LIN {X 0,Y 578.612,Z 1192.309,A -85,B 0,C 180,E1 8897.557,E2 8897.557} C_VEL
LIN {X 0,Y 578.237,Z 1202.22,A -85,B 0,C 180,E1 8901.735,E2 8901.735} C_VEL
LIN {X 0,Y 578.097,Z 1207.67,A -85,B 0,C 180,E1 8905.502,E2 8905.502} C_VEL
LIN {X 0,Y 578.168,Z 1210,A -85,B 0,C 180,E1 8909.999,E2 8909.999} C_VEL
LIN {X 0,Y 578.088,Z 1207.673,A -85,B 0,C 180,E1 8914.497,E2 8914.497} C_VEL
LIN {X 0,Y 578.267,Z 1200.684,A -85,B 0,C 180,E1 8919.02,E2 8919.02} C_VEL
LIN {X 0,Y 578.858,Z 1188.879,A -85,B 0,C 180,E1 8923.588,E2 8923.588} C_VEL
LIN {X 0,Y 580.238,Z 1171.703,A -85,B 0,C 180,E1 8928.21,E2 8928.21} C_VEL
LIN {X 0,Y 582.752,Z 1146.922,A -85,B 0,C 180,E1 8933.18,E2 8933.18} C_VEL
LIN {X 0,Y 586.408,Z 1118.128,A -85,B 0,C 180,E1 8937.635,E2 8937.635} C_VEL
LIN {X 0,Y 591.463,Z 1084.189,A -85,B 0,C 180,E1 8941.799,E2 8941.799} C_VEL
LIN {X 0,Y 597.246,Z 1046.532,A -85,B 0,C 180,E1 8945.448,E2 8945.448} C_VEL
LIN {X 0,Y 603.563,Z 1005.363,A -85,B 0,C 180,E1 8948.616,E2 8948.616} C_VEL
LIN {X 0,Y 609.873,Z 959.425,A -85,B 0,C 180,E1 8951.318,E2 8951.318} C_VEL
LIN {X 0,Y 614.972,Z 913.089,A -85,B 0,C 180,E1 8953.312,E2 8953.312} C_VEL
LIN {X 0,Y 619.146,Z 862.515,A -85,B 0,C 180,E1 8954.794,E2 8954.794} C_VEL
LIN {X 0,Y 620.72,Z 823.615,A -85,B 0,C 180,E1 8955.571,E2 8955.571} C_VEL
LIN {X 0,Y 587.125,Z 766.876,A -85,B 0,C 180,E1 8959.714,E2 8959.714} C_VEL
LIN {X 0,Y 577.318,Z 751.271,A -85,B 0,C 180,E1 8961.134,E2 8961.134} C_VEL
LIN {X 0,Y 577.129,Z 749.56,A -85,B 0,C 180,E1 8961.259,E2 8961.259} C_VEL
LIN {X 0,Y 577.17,Z 749.56,A -85,B 0,C 180,E1 8966.909,E2 8966.909} C_VEL
LIN {X 0,Y 577.189,Z 749.56,A -85,B 0,C 180,E1 8972.89,E2 8972.89} C_VEL
LIN {X 0,Y 577.364,Z 749.56,A -85,B 0,C 180,E1 8978.509,E2 8978.509} C_VEL
LIN {X 0,Y 577.572,Z 749.56,A -85,B 0,C 180,E1 8983.278,E2 8983.278} C_VEL
LIN {X 0,Y 577.694,Z 749.56,A -85,B 0,C 180,E1 8987.925,E2 8987.925} C_VEL
LIN {X 0,Y 577.893,Z 749.56,A -85,B 0,C 180,E1 8993.538,E2 8993.538} C_VEL
LIN {X 0,Y 578.167,Z 749.56,A -85,B 0,C 180,E1 8998.506,E2 8998.506} C_VEL
LIN {X 0,Y 577.98,Z 749.56,A -85,B 0,C 180,E1 9004.503,E2 9004.503} C_VEL
LIN {X 0,Y 577.846,Z 749.56,A -85,B 0,C 180,E1 9009.032,E2 9009.032} C_VEL
LIN {X 0,Y 577.48,Z 749.56,A -85,B 0,C 180,E1 9014.491,E2 9014.491} C_VEL
LIN {X 0,Y 577.308,Z 749.56,A -85,B 0,C 180,E1 9019.899,E2 9019.899} C_VEL
LIN {X 0,Y 577.195,Z 749.56,A -85,B 0,C 180,E1 9024.77,E2 9024.77} C_VEL
LIN {X 0,Y 577.119,Z 749.56,A -85,B 0,C 180,E1 9030.225,E2 9030.225} C_VEL
LIN {X 0,Y 577.219,Z 749.952,A -85,B 0,C 180,E1 9034.568,E2 9034.568} C_VEL
LIN {X 0,Y 579.814,Z 755.423,A -85,B 0,C 180,E1 9034.992,E2 9034.992} C_VEL
LIN {X 0,Y 601.046,Z 789.481,A -85,B 0,C 180,E1 9038.031,E2 9038.031} C_VEL
LIN {X 0,Y 614.345,Z 817.609,A -85,B 0,C 180,E1 9040.099,E2 9040.099} C_VEL
LIN {X 0,Y 610.546,Z 862.835,A -85,B 0,C 180,E1 9041.509,E2 9041.509} C_VEL
LIN {X 0,Y 605.594,Z 905.044,A -85,B 0,C 180,E1 9043.417,E2 9043.417} C_VEL
LIN {X 0,Y 600.085,Z 944.792,A -85,B 0,C 180,E1 9045.805,E2 9045.805} C_VEL
LIN {X 0,Y 593.877,Z 985.069,A -85,B 0,C 180,E1 9049.002,E2 9049.002} C_VEL
LIN {X 0,Y 588.198,Z 1022.822,A -85,B 0,C 180,E1 9052.896,E2 9052.896} C_VEL
LIN {X 0,Y 584.217,Z 1052.857,A -85,B 0,C 180,E1 9056.744,E2 9056.744} C_VEL
LIN {X 0,Y 581.273,Z 1079.147,A -85,B 0,C 180,E1 9061.041,E2 9061.041} C_VEL
LIN {X 0,Y 579.471,Z 1099.154,A -85,B 0,C 180,E1 9065.34,E2 9065.34} C_VEL
LIN {X 0,Y 578.595,Z 1114.303,A -85,B 0,C 180,E1 9069.756,E2 9069.756} C_VEL
LIN {X 0,Y 578.124,Z 1124.044,A -85,B 0,C 180,E1 9074.071,E2 9074.071} C_VEL
LIN {X 0,Y 577.881,Z 1128.776,A -85,B 0,C 180,E1 9077.926,E2 9077.926} C_VEL
LIN {X 0,Y 578.053,Z 1129.657,A -85,B 0,C 180,E1 9082.49,E2 9082.49} C_VEL
LIN {X 0,Y 578.256,Z 1125.379,A -85,B 0,C 180,E1 9087.005,E2 9087.005} C_VEL
LIN {X 0,Y 578.486,Z 1116.064,A -85,B 0,C 180,E1 9091.498,E2 9091.498} C_VEL
LIN {X 0,Y 579.246,Z 1102.955,A -85,B 0,C 180,E1 9095.615,E2 9095.615} C_VEL
LIN {X 0,Y 580.791,Z 1083.025,A -85,B 0,C 180,E1 9100.116,E2 9100.116} C_VEL
LIN {X 0,Y 583.365,Z 1059.112,A -85,B 0,C 180,E1 9104.247,E2 9104.247} C_VEL
LIN {X 0,Y 587.673,Z 1026.88,A -85,B 0,C 180,E1 9108.555,E2 9108.555} C_VEL
LIN {X 0,Y 593.59,Z 986.738,A -85,B 0,C 180,E1 9112.746,E2 9112.746} C_VEL
LIN {X 0,Y 599.698,Z 946.386,A -85,B 0,C 180,E1 9115.968,E2 9115.968} C_VEL
LIN {X 0,Y 605.16,Z 906.666,A -85,B 0,C 180,E1 9118.383,E2 9118.383} C_VEL
LIN {X 0,Y 610.26,Z 863.781,A -85,B 0,C 180,E1 9120.324,E2 9120.324} C_VEL
LIN {X 0,Y 613.896,Z 820.422,A -85,B 0,C 180,E1 9121.706,E2 9121.706} C_VEL
LIN {X 0,Y 612.931,Z 814.925,A -85,B 0,C 180,E1 9121.963,E2 9121.963} C_VEL
LIN {X 0,Y 599.509,Z 787.876,A -85,B 0,C 180,E1 9123.901,E2 9123.901} C_VEL
LIN {X 0,Y 577.285,Z 750.933,A -85,B 0,C 180,E1 9126.769,E2 9126.769} C_VEL
LIN {X 0,Y 577.172,Z 749.56,A -85,B 0,C 180,E1 9126.863,E2 9126.863} C_VEL
LIN {X 0,Y 577.186,Z 749.56,A -85,B 0,C 180,E1 9132.9,E2 9132.9} C_VEL
LIN {X 0,Y 577.153,Z 749.56,A -85,B 0,C 180,E1 9139.107,E2 9139.107} C_VEL
LIN {X 0,Y 577.103,Z 749.56,A -85,B 0,C 180,E1 9144.82,E2 9144.82} C_VEL
LIN {X 0,Y 577.103,Z 749.56,A -85,B 0,C 180,E1 9150.159,E2 9150.159} C_VEL
LIN {X 0,Y 577.201,Z 749.56,A -85,B 0,C 180,E1 9155.231,E2 9155.231} C_VEL
LIN {X 0,Y 577.331,Z 749.56,A -85,B 0,C 180,E1 9160.44,E2 9160.44} C_VEL
LIN {X 0,Y 577.534,Z 749.56,A -85,B 0,C 180,E1 9166.375,E2 9166.375} C_VEL
LIN {X 0,Y 577.842,Z 749.56,A -85,B 0,C 180,E1 9170.968,E2 9170.968} C_VEL
LIN {X 0,Y 578.111,Z 749.56,A -85,B 0,C 180,E1 9176.999,E2 9176.999} C_VEL
LIN {X 0,Y 578.183,Z 749.56,A -85,B 0,C 180,E1 9181.494,E2 9181.494} C_VEL
LIN {X 0,Y 577.908,Z 749.56,A -85,B 0,C 180,E1 9187.508,E2 9187.508} C_VEL
LIN {X 0,Y 577.699,Z 749.56,A -85,B 0,C 180,E1 9193.612,E2 9193.612} C_VEL
LIN {X 0,Y 577.611,Z 749.56,A -85,B 0,C 180,E1 9198.293,E2 9198.293} C_VEL
LIN {X 0,Y 577.4,Z 749.56,A -85,B 0,C 180,E1 9203.651,E2 9203.651} C_VEL
LIN {X 0,Y 577.382,Z 749.56,A -85,B 0,C 180,E1 9208.102,E2 9208.102} C_VEL
LIN {X 0,Y 577.242,Z 749.56,A -85,B 0,C 180,E1 9213.346,E2 9213.346} C_VEL
LIN {X 0,Y 577.164,Z 749.56,A -85,B 0,C 180,E1 9218.983,E2 9218.983} C_VEL
LIN {X 0,Y 579.391,Z 755.018,A -85,B 0,C 180,E1 9219.32,E2 9219.32} C_VEL
LIN {X 0,Y 610.577,Z 806.083,A -85,B 0,C 180,E1 9223.218,E2 9223.218} C_VEL
LIN {X 0,Y 621.286,Z 825.092,A -85,B 0,C 180,E1 9224.485,E2 9224.485} C_VEL
LIN {X 0,Y 618.48,Z 874.739,A -85,B 0,C 180,E1 9225.498,E2 9225.498} C_VEL
LIN {X 0,Y 614.01,Z 922.392,A -85,B 0,C 180,E1 9227.039,E2 9227.039} C_VEL
LIN {X 0,Y 613.212,Z 931.376,A -85,B 0,C 180,E1 9227.398,E2 9227.398} C_VEL
LIN {X 0,Y 608.294,Z 947.479,A -85,B 0,C 180,E1 9227.866,E2 9227.866} C_VEL
LIN {X 0,Y 603.135,Z 963.24,A -85,B 0,C 180,E1 9228.403,E2 9228.403} C_VEL
LIN {X 0,Y 597.496,Z 1003.581,A -85,B 0,C 180,E1 9230.781,E2 9230.781} C_VEL
LIN {X 0,Y 591.158,Z 1043.01,A -85,B 0,C 180,E1 9233.785,E2 9233.785} C_VEL
LIN {X 0,Y 584.765,Z 1082.334,A -85,B 0,C 180,E1 9237.573,E2 9237.573} C_VEL
LIN {X 0,Y 579.229,Z 1116.9,A -85,B 0,C 180,E1 9241.815,E2 9241.815} C_VEL
LIN {X 0,Y 575.32,Z 1145.203,A -85,B 0,C 180,E1 9246.181,E2 9246.181} C_VEL
LIN {X 0,Y 572.667,Z 1168.231,A -85,B 0,C 180,E1 9250.74,E2 9250.74} C_VEL
LIN {X 0,Y 571.23,Z 1186.567,A -85,B 0,C 180,E1 9255.501,E2 9255.501} C_VEL
LIN {X 0,Y 570.523,Z 1199.103,A -85,B 0,C 180,E1 9260.086,E2 9260.086} C_VEL
LIN {X 0,Y 570.308,Z 1205.908,A -85,B 0,C 180,E1 9263.915,E2 9263.915} C_VEL
LIN {X 0,Y 570.149,Z 1209.667,A -85,B 0,C 180,E1 9268.48,E2 9268.48} C_VEL
LIN {X 0,Y 570.3,Z 1208.914,A -85,B 0,C 180,E1 9273.037,E2 9273.037} C_VEL
LIN {X 0,Y 570.311,Z 1203.554,A -85,B 0,C 180,E1 9277.612,E2 9277.612} C_VEL
LIN {X 0,Y 570.709,Z 1193.421,A -85,B 0,C 180,E1 9282.229,E2 9282.229} C_VEL
LIN {X 0,Y 571.785,Z 1178.004,A -85,B 0,C 180,E1 9286.9,E2 9286.9} C_VEL
LIN {X 0,Y 573.906,Z 1156.975,A -85,B 0,C 180,E1 9291.63,E2 9291.63} C_VEL
LIN {X 0,Y 577.264,Z 1130.743,A -85,B 0,C 180,E1 9296.17,E2 9296.17} C_VEL
LIN {X 0,Y 582.138,Z 1098.258,A -85,B 0,C 180,E1 9300.604,E2 9300.604} C_VEL
LIN {X 0,Y 588.075,Z 1061.38,A -85,B 0,C 180,E1 9304.559,E2 9304.559} C_VEL
LIN {X 0,Y 594.538,Z 1021.722,A -85,B 0,C 180,E1 9307.94,E2 9307.94} C_VEL
LIN {X 0,Y 601.245,Z 978.007,A -85,B 0,C 180,E1 9310.802,E2 9310.802} C_VEL
LIN {X 0,Y 606.913,Z 932.395,A -85,B 0,C 180,E1 9313.024,E2 9313.024} C_VEL
LIN {X 0,Y 611.296,Z 887.394,A -85,B 0,C 180,E1 9314.618,E2 9314.618} C_VEL
LIN {X 0,Y 614.809,Z 838.477,A -85,B 0,C 180,E1 9315.774,E2 9315.774} C_VEL
LIN {X 0,Y 614.638,Z 826.617,A -85,B 0,C 180,E1 9316.032,E2 9316.032} C_VEL
LIN {X 0,Y 582.329,Z 771.526,A -85,B 0,C 180,E1 9320.165,E2 9320.165} C_VEL
LIN {X 0,Y 571.112,Z 754.658,A -85,B 0,C 180,E1 9321.827,E2 9321.827} C_VEL
LIN {X 0,Y 569.234,Z 749.56,A -85,B 0,C 180,E1 9322.219,E2 9322.219} C_VEL
LIN {X 0,Y 569.252,Z 749.56,A -85,B 0,C 180,E1 9328.152,E2 9328.152} C_VEL
LIN {X 0,Y 569.31,Z 749.56,A -85,B 0,C 180,E1 9333.181,E2 9333.181} C_VEL
LIN {X 0,Y 569.446,Z 749.56,A -85,B 0,C 180,E1 9338.245,E2 9338.245} C_VEL
LIN {X 0,Y 569.635,Z 749.56,A -85,B 0,C 180,E1 9343.038,E2 9343.038} C_VEL
LIN {X 0,Y 569.819,Z 749.56,A -85,B 0,C 180,E1 9348.874,E2 9348.874} C_VEL
LIN {X 0,Y 570.05,Z 749.56,A -85,B 0,C 180,E1 9353.917,E2 9353.917} C_VEL
LIN {X 0,Y 570.266,Z 749.56,A -85,B 0,C 180,E1 9360.004,E2 9360.004} C_VEL
LIN {X 0,Y 570.07,Z 749.56,A -85,B 0,C 180,E1 9364.565,E2 9364.565} C_VEL
LIN {X 0,Y 569.921,Z 749.56,A -85,B 0,C 180,E1 9369.158,E2 9369.158} C_VEL
LIN {X 0,Y 569.615,Z 749.56,A -85,B 0,C 180,E1 9373.818,E2 9373.818} C_VEL
LIN {X 0,Y 569.384,Z 749.56,A -85,B 0,C 180,E1 9378.576,E2 9378.576} C_VEL
LIN {X 0,Y 569.302,Z 749.56,A -85,B 0,C 180,E1 9383.468,E2 9383.468} C_VEL
LIN {X 0,Y 569.204,Z 749.56,A -85,B 0,C 180,E1 9388.828,E2 9388.828} C_VEL
LIN {X 0,Y 569.282,Z 749.594,A -85,B 0,C 180,E1 9393.55,E2 9393.55} C_VEL
LIN {X 0,Y 571.523,Z 755.068,A -85,B 0,C 180,E1 9393.95,E2 9393.95} C_VEL
LIN {X 0,Y 589.479,Z 782.711,A -85,B 0,C 180,E1 9396.648,E2 9396.648} C_VEL
LIN {X 0,Y 605.75,Z 813.927,A -85,B 0,C 180,E1 9399.164,E2 9399.164} C_VEL
LIN {X 0,Y 608.425,Z 822.45,A -85,B 0,C 180,E1 9399.699,E2 9399.699} C_VEL
LIN {X 0,Y 604.318,Z 866.169,A -85,B 0,C 180,E1 9401.115,E2 9401.115} C_VEL
LIN {X 0,Y 598.886,Z 910.311,A -85,B 0,C 180,E1 9403.176,E2 9403.176} C_VEL
LIN {X 0,Y 592.946,Z 950.211,A -85,B 0,C 180,E1 9405.687,E2 9405.687} C_VEL
LIN {X 0,Y 586.591,Z 989.264,A -85,B 0,C 180,E1 9408.889,E2 9408.889} C_VEL
LIN {X 0,Y 580.689,Z 1025.536,A -85,B 0,C 180,E1 9412.786,E2 9412.786} C_VEL
LIN {X 0,Y 575.878,Z 1059.375,A -85,B 0,C 180,E1 9417.383,E2 9417.383} C_VEL
LIN {X 0,Y 573.067,Z 1083.698,A -85,B 0,C 180,E1 9421.665,E2 9421.665} C_VEL
LIN {X 0,Y 571.421,Z 1103.026,A -85,B 0,C 180,E1 9426.107,E2 9426.107} C_VEL
LIN {X 0,Y 570.606,Z 1117.129,A -85,B 0,C 180,E1 9430.693,E2 9430.693} C_VEL
LIN {X 0,Y 570.191,Z 1125.995,A -85,B 0,C 180,E1 9435.211,E2 9435.211} C_VEL
LIN {X 0,Y 569.984,Z 1129.637,A -85,B 0,C 180,E1 9439.306,E2 9439.306} C_VEL
LIN {X 0,Y 570.162,Z 1128.85,A -85,B 0,C 180,E1 9443.915,E2 9443.915} C_VEL
LIN {X 0,Y 570.299,Z 1123.147,A -85,B 0,C 180,E1 9448.482,E2 9448.482} C_VEL
LIN {X 0,Y 570.789,Z 1113.278,A -85,B 0,C 180,E1 9452.656,E2 9452.656} C_VEL
LIN {X 0,Y 571.884,Z 1097.491,A -85,B 0,C 180,E1 9457.211,E2 9457.211} C_VEL
LIN {X 0,Y 574.022,Z 1075.686,A -85,B 0,C 180,E1 9461.773,E2 9461.773} C_VEL
LIN {X 0,Y 577.236,Z 1049.762,A -85,B 0,C 180,E1 9465.955,E2 9465.955} C_VEL
LIN {X 0,Y 582.581,Z 1013.881,A -85,B 0,C 180,E1 9470.477,E2 9470.477} C_VEL
LIN {X 0,Y 588.507,Z 977.222,A -85,B 0,C 180,E1 9474.072,E2 9474.072} C_VEL
LIN {X 0,Y 594.407,Z 938.894,A -85,B 0,C 180,E1 9476.981,E2 9476.981} C_VEL
LIN {X 0,Y 600.477,Z 895.788,A -85,B 0,C 180,E1 9479.464,E2 9479.464} C_VEL
LIN {X 0,Y 605.681,Z 850.137,A -85,B 0,C 180,E1 9481.335,E2 9481.335} C_VEL
LIN {X 0,Y 607.753,Z 819.864,A -85,B 0,C 180,E1 9482.278,E2 9482.278} C_VEL
LIN {X 0,Y 595.074,Z 793.605,A -85,B 0,C 180,E1 9484.196,E2 9484.196} C_VEL
LIN {X 0,Y 569.437,Z 751.318,A -85,B 0,C 180,E1 9487.595,E2 9487.595} C_VEL
LIN {X 0,Y 569.233,Z 749.56,A -85,B 0,C 180,E1 9487.784,E2 9487.784} C_VEL
LIN {X 0,Y 569.194,Z 749.56,A -85,B 0,C 180,E1 9493.652,E2 9493.652} C_VEL
LIN {X 0,Y 569.167,Z 749.56,A -85,B 0,C 180,E1 9498.407,E2 9498.407} C_VEL
LIN {X 0,Y 569.217,Z 749.56,A -85,B 0,C 180,E1 9504.258,E2 9504.258} C_VEL
LIN {X 0,Y 569.192,Z 749.56,A -85,B 0,C 180,E1 9509.701,E2 9509.701} C_VEL
LIN {X 0,Y 569.248,Z 749.56,A -85,B 0,C 180,E1 9514.861,E2 9514.861} C_VEL
LIN {X 0,Y 569.364,Z 749.56,A -85,B 0,C 180,E1 9519.812,E2 9519.812} C_VEL
LIN {X 0,Y 569.496,Z 749.56,A -85,B 0,C 180,E1 9524.608,E2 9524.608} C_VEL
LIN {X 0,Y 569.819,Z 749.56,A -85,B 0,C 180,E1 9529.297,E2 9529.297} C_VEL
LIN {X 0,Y 570.017,Z 749.56,A -85,B 0,C 180,E1 9533.908,E2 9533.908} C_VEL
LIN {X 0,Y 570.138,Z 749.56,A -85,B 0,C 180,E1 9538.477,E2 9538.477} C_VEL
LIN {X 0,Y 570.069,Z 749.56,A -85,B 0,C 180,E1 9543.035,E2 9543.035} C_VEL
LIN {X 0,Y 569.99,Z 749.56,A -85,B 0,C 180,E1 9547.613,E2 9547.613} C_VEL
LIN {X 0,Y 569.785,Z 749.56,A -85,B 0,C 180,E1 9553.805,E2 9553.805} C_VEL
LIN {X 0,Y 569.686,Z 749.56,A -85,B 0,C 180,E1 9558.557,E2 9558.557} C_VEL
LIN {X 0,Y 569.509,Z 749.56,A -85,B 0,C 180,E1 9563.45,E2 9563.45} C_VEL
LIN {X 0,Y 569.389,Z 749.56,A -85,B 0,C 180,E1 9568.858,E2 9568.858} C_VEL
LIN {X 0,Y 569.253,Z 749.56,A -85,B 0,C 180,E1 9574.621,E2 9574.621} C_VEL
LIN {X 0,Y 569.31,Z 750.309,A -85,B 0,C 180,E1 9578.161,E2 9578.161} C_VEL
LIN {X 0,Y 572.281,Z 755.784,A -85,B 0,C 180,E1 9578.584,E2 9578.584} C_VEL
LIN {X 0,Y 606.158,Z 811.799,A -85,B 0,C 180,E1 9582.908,E2 9582.908} C_VEL
LIN {X 0,Y 615.297,Z 827.805,A -85,B 0,C 180,E1 9584.02,E2 9584.02} C_VEL
LIN {X 0,Y 612.316,Z 876.778,A -85,B 0,C 180,E1 9585.064,E2 9585.064} C_VEL
LIN {X 0,Y 607.591,Z 924.963,A -85,B 0,C 180,E1 9586.663,E2 9586.663} C_VEL
LIN {X 0,Y 603.135,Z 963.24,A -85,B 0,C 180,E1 9588.403,E2 9588.403} C_VEL
LIN {X 0,Y 598,Z 978.76,A -85,B 0,C 180,E1 9589.009,E2 9589.009} C_VEL
LIN {X 0,Y 592.579,Z 993.901,A -85,B 0,C 180,E1 9589.68,E2 9589.68} C_VEL
LIN {X 0,Y 586.197,Z 1032.86,A -85,B 0,C 180,E1 9592.455,E2 9592.455} C_VEL
LIN {X 0,Y 579.745,Z 1070.845,A -85,B 0,C 180,E1 9595.915,E2 9595.915} C_VEL
LIN {X 0,Y 573.522,Z 1107.345,A -85,B 0,C 180,E1 9600.13,E2 9600.13} C_VEL
LIN {X 0,Y 569.067,Z 1136.294,A -85,B 0,C 180,E1 9604.343,E2 9604.343} C_VEL
LIN {X 0,Y 565.606,Z 1162.666,A -85,B 0,C 180,E1 9609.235,E2 9609.235} C_VEL
LIN {X 0,Y 563.725,Z 1181.011,A -85,B 0,C 180,E1 9613.652,E2 9613.652} C_VEL
LIN {X 0,Y 562.769,Z 1195.153,A -85,B 0,C 180,E1 9618.284,E2 9618.284} C_VEL
LIN {X 0,Y 562.455,Z 1204.876,A -85,B 0,C 180,E1 9623.133,E2 9623.133} C_VEL
LIN {X 0,Y 562.361,Z 1208.909,A -85,B 0,C 180,E1 9626.919,E2 9626.919} C_VEL
LIN {X 0,Y 562.506,Z 1209.667,A -85,B 0,C 180,E1 9631.539,E2 9631.539} C_VEL
LIN {X 0,Y 562.41,Z 1205.831,A -85,B 0,C 180,E1 9636.23,E2 9636.23} C_VEL
LIN {X 0,Y 562.718,Z 1197.317,A -85,B 0,C 180,E1 9640.834,E2 9640.834} C_VEL
LIN {X 0,Y 563.546,Z 1183.708,A -85,B 0,C 180,E1 9645.553,E2 9645.553} C_VEL
LIN {X 0,Y 565.132,Z 1166.494,A -85,B 0,C 180,E1 9649.933,E2 9649.933} C_VEL
LIN {X 0,Y 568.012,Z 1142.832,A -85,B 0,C 180,E1 9654.562,E2 9654.562} C_VEL
LIN {X 0,Y 572.688,Z 1112.559,A -85,B 0,C 180,E1 9659.18,E2 9659.18} C_VEL
LIN {X 0,Y 578.359,Z 1078.518,A -85,B 0,C 180,E1 9663.276,E2 9663.276} C_VEL
LIN {X 0,Y 585.156,Z 1039.262,A -85,B 0,C 180,E1 9667.024,E2 9667.024} C_VEL
LIN {X 0,Y 591.517,Z 1000.569,A -85,B 0,C 180,E1 9669.905,E2 9669.905} C_VEL
LIN {X 0,Y 597.952,Z 953.868,A -85,B 0,C 180,E1 9672.532,E2 9672.532} C_VEL
LIN {X 0,Y 603.268,Z 906.93,A -85,B 0,C 180,E1 9674.488,E2 9674.488} C_VEL
LIN {X 0,Y 607.841,Z 855.273,A -85,B 0,C 180,E1 9675.951,E2 9675.951} C_VEL
LIN {X 0,Y 609.068,Z 830.48,A -85,B 0,C 180,E1 9676.444,E2 9676.444} C_VEL
LIN {X 0,Y 577.572,Z 776.18,A -85,B 0,C 180,E1 9680.624,E2 9680.624} C_VEL
LIN {X 0,Y 563.661,Z 755.147,A -85,B 0,C 180,E1 9682.777,E2 9682.777} C_VEL
LIN {X 0,Y 561.297,Z 749.56,A -85,B 0,C 180,E1 9683.323,E2 9683.323} C_VEL
LIN {X 0,Y 561.314,Z 749.56,A -85,B 0,C 180,E1 9689.482,E2 9689.482} C_VEL
LIN {X 0,Y 561.42,Z 749.56,A -85,B 0,C 180,E1 9694.495,E2 9694.495} C_VEL
LIN {X 0,Y 561.587,Z 749.56,A -85,B 0,C 180,E1 9700.351,E2 9700.351} C_VEL
LIN {X 0,Y 561.838,Z 749.56,A -85,B 0,C 180,E1 9705.996,E2 9705.996} C_VEL
LIN {X 0,Y 562.005,Z 749.56,A -85,B 0,C 180,E1 9710.72,E2 9710.72} C_VEL
LIN {X 0,Y 562.189,Z 749.56,A -85,B 0,C 180,E1 9715.379,E2 9715.379} C_VEL
LIN {X 0,Y 562.365,Z 749.56,A -85,B 0,C 180,E1 9720.004,E2 9720.004} C_VEL
LIN {X 0,Y 562.159,Z 749.56,A -85,B 0,C 180,E1 9724.63,E2 9724.63} C_VEL
LIN {X 0,Y 562.006,Z 749.56,A -85,B 0,C 180,E1 9729.289,E2 9729.289} C_VEL
LIN {X 0,Y 561.66,Z 749.56,A -85,B 0,C 180,E1 9734.407,E2 9734.407} C_VEL
LIN {X 0,Y 561.446,Z 749.56,A -85,B 0,C 180,E1 9740.486,E2 9740.486} C_VEL
LIN {X 0,Y 561.357,Z 749.56,A -85,B 0,C 180,E1 9745.518,E2 9745.518} C_VEL
LIN {X 0,Y 561.29,Z 749.56,A -85,B 0,C 180,E1 9751.526,E2 9751.526} C_VEL
LIN {X 0,Y 561.297,Z 749.56,A -85,B 0,C 180,E1 9752.472,E2 9752.472} C_VEL
LIN {X 0,Y 563.51,Z 755.009,A -85,B 0,C 180,E1 9752.89,E2 9752.89} C_VEL
LIN {X 0,Y 577.76,Z 775.916,A -85,B 0,C 180,E1 9755.134,E2 9755.134} C_VEL
LIN {X 0,Y 595.276,Z 806.94,A -85,B 0,C 180,E1 9757.886,E2 9757.886} C_VEL
LIN {X 0,Y 602.732,Z 824.081,A -85,B 0,C 180,E1 9759.2,E2 9759.2} C_VEL
LIN {X 0,Y 598.408,Z 867.609,A -85,B 0,C 180,E1 9760.636,E2 9760.636} C_VEL
LIN {X 0,Y 592.864,Z 910.622,A -85,B 0,C 180,E1 9762.665,E2 9762.665} C_VEL
LIN {X 0,Y 586.622,Z 950.54,A -85,B 0,C 180,E1 9765.188,E2 9765.188} C_VEL
LIN {X 0,Y 580.114,Z 988.793,A -85,B 0,C 180,E1 9768.338,E2 9768.338} C_VEL
LIN {X 0,Y 573.941,Z 1024.495,A -85,B 0,C 180,E1 9772.182,E2 9772.182} C_VEL
LIN {X 0,Y 568.989,Z 1055.093,A -85,B 0,C 180,E1 9776.407,E2 9776.407} C_VEL
LIN {X 0,Y 565.873,Z 1079.951,A -85,B 0,C 180,E1 9780.63,E2 9780.63} C_VEL
LIN {X 0,Y 563.785,Z 1100.396,A -85,B 0,C 180,E1 9785.218,E2 9785.218} C_VEL
LIN {X 0,Y 562.873,Z 1114.699,A -85,B 0,C 180,E1 9789.574,E2 9789.574} C_VEL
LIN {X 0,Y 562.349,Z 1124.877,A -85,B 0,C 180,E1 9794.413,E2 9794.413} C_VEL
LIN {X 0,Y 562.087,Z 1129.608,A -85,B 0,C 180,E1 9799.154,E2 9799.154} C_VEL
LIN {X 0,Y 562.254,Z 1128.822,A -85,B 0,C 180,E1 9803.998,E2 9803.998} C_VEL
LIN {X 0,Y 562.403,Z 1123.372,A -85,B 0,C 180,E1 9808.461,E2 9808.461} C_VEL
LIN {X 0,Y 562.902,Z 1113.654,A -85,B 0,C 180,E1 9812.693,E2 9812.693} C_VEL
LIN {X 0,Y 564.07,Z 1097.98,A -85,B 0,C 180,E1 9817.315,E2 9817.315} C_VEL
LIN {X 0,Y 566.182,Z 1077.441,A -85,B 0,C 180,E1 9821.743,E2 9821.743} C_VEL
LIN {X 0,Y 569.857,Z 1049.36,A -85,B 0,C 180,E1 9826.365,E2 9826.365} C_VEL
LIN {X 0,Y 575.388,Z 1015.913,A -85,B 0,C 180,E1 9830.731,E2 9830.731} C_VEL
LIN {X 0,Y 581.602,Z 979.378,A -85,B 0,C 180,E1 9834.383,E2 9834.383} C_VEL
LIN {X 0,Y 587.752,Z 941.688,A -85,B 0,C 180,E1 9837.312,E2 9837.312} C_VEL
LIN {X 0,Y 594.335,Z 897.041,A -85,B 0,C 180,E1 9839.928,E2 9839.928} C_VEL
LIN {X 0,Y 599.696,Z 852.103,A -85,B 0,C 180,E1 9841.79,E2 9841.79} C_VEL
LIN {X 0,Y 601.685,Z 822.463,A -85,B 0,C 180,E1 9842.75,E2 9842.75} C_VEL
LIN {X 0,Y 587.274,Z 793.511,A -85,B 0,C 180,E1 9844.954,E2 9844.954} C_VEL
LIN {X 0,Y 561.404,Z 750.508,A -85,B 0,C 180,E1 9848.496,E2 9848.496} C_VEL
LIN {X 0,Y 561.343,Z 749.56,A -85,B 0,C 180,E1 9848.669,E2 9848.669} C_VEL
LIN {X 0,Y 561.299,Z 749.56,A -85,B 0,C 180,E1 9854.426,E2 9854.426} C_VEL
LIN {X 0,Y 561.223,Z 749.56,A -85,B 0,C 180,E1 9859.736,E2 9859.736} C_VEL
LIN {X 0,Y 561.294,Z 749.56,A -85,B 0,C 180,E1 9865.566,E2 9865.566} C_VEL
LIN {X 0,Y 561.264,Z 749.56,A -85,B 0,C 180,E1 9871.006,E2 9871.006} C_VEL
LIN {X 0,Y 561.376,Z 749.56,A -85,B 0,C 180,E1 9876.239,E2 9876.239} C_VEL
LIN {X 0,Y 561.448,Z 749.56,A -85,B 0,C 180,E1 9881.152,E2 9881.152} C_VEL
LIN {X 0,Y 561.671,Z 749.56,A -85,B 0,C 180,E1 9885.983,E2 9885.983} C_VEL
LIN {X 0,Y 562.005,Z 749.56,A -85,B 0,C 180,E1 9890.711,E2 9890.711} C_VEL
LIN {X 0,Y 562.293,Z 749.56,A -85,B 0,C 180,E1 9896.915,E2 9896.915} C_VEL
LIN {X 0,Y 562.368,Z 749.56,A -85,B 0,C 180,E1 9901.536,E2 9901.536} C_VEL
LIN {X 0,Y 562.08,Z 749.56,A -85,B 0,C 180,E1 9907.721,E2 9907.721} C_VEL
LIN {X 0,Y 561.884,Z 749.56,A -85,B 0,C 180,E1 9912.42,E2 9912.42} C_VEL
LIN {X 0,Y 561.816,Z 749.56,A -85,B 0,C 180,E1 9917.206,E2 9917.206} C_VEL
LIN {X 0,Y 561.638,Z 749.56,A -85,B 0,C 180,E1 9922.124,E2 9922.124} C_VEL
LIN {X 0,Y 561.528,Z 749.56,A -85,B 0,C 180,E1 9927.368,E2 9927.368} C_VEL
LIN {X 0,Y 561.35,Z 749.56,A -85,B 0,C 180,E1 9932.57,E2 9932.57} C_VEL
LIN {X 0,Y 561.38,Z 749.56,A -85,B 0,C 180,E1 9937.265,E2 9937.265} C_VEL
LIN {X 0,Y 563.756,Z 755.23,A -85,B 0,C 180,E1 9937.642,E2 9937.642} C_VEL
LIN {X 0,Y 594.417,Z 804.941,A -85,B 0,C 180,E1 9941.684,E2 9941.684} C_VEL
LIN {X 0,Y 609.445,Z 831.101,A -85,B 0,C 180,E1 9943.566,E2 9943.566} C_VEL
LIN {X 0,Y 605.951,Z 881.237,A -85,B 0,C 180,E1 9944.691,E2 9944.691} C_VEL
LIN {X 0,Y 601.062,Z 928.661,A -85,B 0,C 180,E1 9946.323,E2 9946.323} C_VEL
LIN {X 0,Y 595.175,Z 974.72,A -85,B 0,C 180,E1 9948.542,E2 9948.542} C_VEL
LIN {X 0,Y 592.579,Z 993.901,A -85,B 0,C 180,E1 9949.68,E2 9949.68} C_VEL
LIN {X 0,Y 586.992,Z 1008.779,A -85,B 0,C 180,E1 9950.406,E2 9950.406} C_VEL
LIN {X 0,Y 581.298,Z 1023.202,A -85,B 0,C 180,E1 9951.206,E2 9951.206} C_VEL
LIN {X 0,Y 574.745,Z 1060.533,A -85,B 0,C 180,E1 9954.428,E2 9954.428} C_VEL
LIN {X 0,Y 568.08,Z 1097.562,A -85,B 0,C 180,E1 9958.457,E2 9958.457} C_VEL
LIN {X 0,Y 562.494,Z 1130.449,A -85,B 0,C 180,E1 9963.041,E2 9963.041} C_VEL
LIN {X 0,Y 558.657,Z 1156.976,A -85,B 0,C 180,E1 9967.747,E2 9967.747} C_VEL
LIN {X 0,Y 556.326,Z 1177.995,A -85,B 0,C 180,E1 9972.614,E2 9972.614} C_VEL
LIN {X 0,Y 555.018,Z 1193.416,A -85,B 0,C 180,E1 9977.419,E2 9977.419} C_VEL
LIN {X 0,Y 554.547,Z 1203.545,A -85,B 0,C 180,E1 9982.168,E2 9982.168} C_VEL
LIN {X 0,Y 554.466,Z 1208.906,A -85,B 0,C 180,E1 9986.875,E2 9986.875} C_VEL
LIN {X 0,Y 554.627,Z 1209.667,A -85,B 0,C 180,E1 9991.56,E2 9991.56} C_VEL
LIN {X 0,Y 554.538,Z 1205.911,A -85,B 0,C 180,E1 9996.257,E2 9996.257} C_VEL
LIN {X 0,Y 554.841,Z 1197.314,A -85,B 0,C 180,E1 10000.99,E2 10000.99} C_VEL
LIN {X 0,Y 555.71,Z 1183.707,A -85,B 0,C 180,E1 10005.778,E2 10005.778} C_VEL
LIN {X 0,Y 557.686,Z 1164.736,A -85,B 0,C 180,E1 10010.624,E2 10010.624} C_VEL
LIN {X 0,Y 560.834,Z 1140.431,A -85,B 0,C 180,E1 10015.323,E2 10015.323} C_VEL
LIN {X 0,Y 565.905,Z 1109.977,A -85,B 0,C 180,E1 10019.949,E2 10019.949} C_VEL
LIN {X 0,Y 572.134,Z 1074.771,A -85,B 0,C 180,E1 10024.132,E2 10024.132} C_VEL
LIN {X 0,Y 578.939,Z 1037.487,A -85,B 0,C 180,E1 10027.665,E2 10027.665} C_VEL
LIN {X 0,Y 585.312,Z 997.916,A -85,B 0,C 180,E1 10030.527,E2 10030.527} C_VEL
LIN {X 0,Y 591.991,Z 951.646,A -85,B 0,C 180,E1 10033.119,E2 10033.119} C_VEL
LIN {X 0,Y 597.537,Z 904.082,A -85,B 0,C 180,E1 10035.079,E2 10035.079} C_VEL
LIN {X 0,Y 602.039,Z 854.566,A -85,B 0,C 180,E1 10036.476,E2 10036.476} C_VEL
LIN {X 0,Y 603.093,Z 833.6,A -85,B 0,C 180,E1 10036.914,E2 10036.914} C_VEL
LIN {X 0,Y 572.381,Z 779.831,A -85,B 0,C 180,E1 10041.174,E2 10041.174} C_VEL
LIN {X 0,Y 556.035,Z 755.418,A -85,B 0,C 180,E1 10043.815,E2 10043.815} C_VEL
LIN {X 0,Y 553.401,Z 750.081,A -85,B 0,C 180,E1 10044.308,E2 10044.308} C_VEL
LIN {X 0,Y 553.336,Z 749.56,A -85,B 0,C 180,E1 10048.747,E2 10048.747} C_VEL
LIN {X 0,Y 553.496,Z 749.56,A -85,B 0,C 180,E1 10054.281,E2 10054.281} C_VEL
LIN {X 0,Y 553.615,Z 749.56,A -85,B 0,C 180,E1 10059.22,E2 10059.22} C_VEL
LIN {X 0,Y 553.839,Z 749.56,A -85,B 0,C 180,E1 10064.17,E2 10064.17} C_VEL
LIN {X 0,Y 554.023,Z 749.56,A -85,B 0,C 180,E1 10069.084,E2 10069.084} C_VEL
LIN {X 0,Y 554.235,Z 749.56,A -85,B 0,C 180,E1 10073.743,E2 10073.743} C_VEL
LIN {X 0,Y 554.488,Z 749.56,A -85,B 0,C 180,E1 10080.004,E2 10080.004} C_VEL
LIN {X 0,Y 554.256,Z 749.56,A -85,B 0,C 180,E1 10084.696,E2 10084.696} C_VEL
LIN {X 0,Y 554.08,Z 749.56,A -85,B 0,C 180,E1 10089.423,E2 10089.423} C_VEL
LIN {X 0,Y 553.785,Z 749.56,A -85,B 0,C 180,E1 10094.221,E2 10094.221} C_VEL
LIN {X 0,Y 553.534,Z 749.56,A -85,B 0,C 180,E1 10099.128,E2 10099.128} C_VEL
LIN {X 0,Y 553.421,Z 749.56,A -85,B 0,C 180,E1 10104.184,E2 10104.184} C_VEL
LIN {X 0,Y 553.373,Z 749.56,A -85,B 0,C 180,E1 10109.447,E2 10109.447} C_VEL
LIN {X 0,Y 553.422,Z 750.37,A -85,B 0,C 180,E1 10111.363,E2 10111.363} C_VEL
LIN {X 0,Y 556.172,Z 755.585,A -85,B 0,C 180,E1 10111.876,E2 10111.876} C_VEL
LIN {X 0,Y 574.693,Z 783.262,A -85,B 0,C 180,E1 10114.928,E2 10114.928} C_VEL
LIN {X 0,Y 591.987,Z 814.965,A -85,B 0,C 180,E1 10117.786,E2 10117.786} C_VEL
LIN {X 0,Y 596.967,Z 827.669,A -85,B 0,C 180,E1 10118.74,E2 10118.74} C_VEL
LIN {X 0,Y 592.158,Z 872.263,A -85,B 0,C 180,E1 10120.276,E2 10120.276} C_VEL
LIN {X 0,Y 586.17,Z 915.89,A -85,B 0,C 180,E1 10122.413,E2 10122.413} C_VEL
LIN {X 0,Y 579.336,Z 956.881,A -85,B 0,C 180,E1 10125.127,E2 10125.127} C_VEL
LIN {X 0,Y 572.836,Z 992.761,A -85,B 0,C 180,E1 10128.209,E2 10128.209} C_VEL
LIN {X 0,Y 566.415,Z 1028.291,A -85,B 0,C 180,E1 10132.15,E2 10132.15} C_VEL
LIN {X 0,Y 561.083,Z 1059.102,A -85,B 0,C 180,E1 10136.616,E2 10136.616} C_VEL
LIN {X 0,Y 557.369,Z 1086.93,A -85,B 0,C 180,E1 10141.783,E2 10141.783} C_VEL
LIN {X 0,Y 555.643,Z 1105.296,A -85,B 0,C 180,E1 10146.351,E2 10146.351} C_VEL
LIN {X 0,Y 554.765,Z 1118.402,A -85,B 0,C 180,E1 10150.922,E2 10150.922} C_VEL
LIN {X 0,Y 554.389,Z 1126.167,A -85,B 0,C 180,E1 10155.159,E2 10155.159} C_VEL
LIN {X 0,Y 554.172,Z 1129.581,A -85,B 0,C 180,E1 10159.038,E2 10159.038} C_VEL
LIN {X 0,Y 554.354,Z 1129.019,A -85,B 0,C 180,E1 10163.741,E2 10163.741} C_VEL
LIN {X 0,Y 554.509,Z 1123.571,A -85,B 0,C 180,E1 10168.439,E2 10168.439} C_VEL
LIN {X 0,Y 555.025,Z 1114.03,A -85,B 0,C 180,E1 10172.732,E2 10172.732} C_VEL
LIN {X 0,Y 556.244,Z 1098.481,A -85,B 0,C 180,E1 10177.418,E2 10177.418} C_VEL
LIN {X 0,Y 558.477,Z 1078.15,A -85,B 0,C 180,E1 10181.907,E2 10181.907} C_VEL
LIN {X 0,Y 562.872,Z 1048.315,A -85,B 0,C 180,E1 10186.976,E2 10186.976} C_VEL
LIN {X 0,Y 568.496,Z 1016.33,A -85,B 0,C 180,E1 10191.175,E2 10191.175} C_VEL
LIN {X 0,Y 575.068,Z 979.732,A -85,B 0,C 180,E1 10194.863,E2 10194.863} C_VEL
LIN {X 0,Y 581.673,Z 941.021,A -85,B 0,C 180,E1 10197.881,E2 10197.881} C_VEL
LIN {X 0,Y 588.268,Z 897.975,A -85,B 0,C 180,E1 10200.411,E2 10200.411} C_VEL
LIN {X 0,Y 593.844,Z 852.664,A -85,B 0,C 180,E1 10202.303,E2 10202.303} C_VEL
LIN {X 0,Y 595.888,Z 825.822,A -85,B 0,C 180,E1 10203.181,E2 10203.181} C_VEL
LIN {X 0,Y 579.952,Z 794.187,A -85,B 0,C 180,E1 10205.667,E2 10205.667} C_VEL
LIN {X 0,Y 555.268,Z 754.686,A -85,B 0,C 180,E1 10209.117,E2 10209.117} C_VEL
LIN {X 0,Y 553.344,Z 749.56,A -85,B 0,C 180,E1 10209.496,E2 10209.496} C_VEL
LIN {X 0,Y 553.395,Z 749.56,A -85,B 0,C 180,E1 10215.233,E2 10215.233} C_VEL
LIN {X 0,Y 553.297,Z 749.56,A -85,B 0,C 180,E1 10221.079,E2 10221.079} C_VEL
LIN {X 0,Y 553.326,Z 749.56,A -85,B 0,C 180,E1 10226.887,E2 10226.887} C_VEL
LIN {X 0,Y 553.358,Z 749.56,A -85,B 0,C 180,E1 10232.333,E2 10232.333} C_VEL
LIN {X 0,Y 553.507,Z 749.56,A -85,B 0,C 180,E1 10238.163,E2 10238.163} C_VEL
LIN {X 0,Y 553.641,Z 749.56,A -85,B 0,C 180,E1 10244.156,E2 10244.156} C_VEL
LIN {X 0,Y 553.999,Z 749.56,A -85,B 0,C 180,E1 10249.105,E2 10249.105} C_VEL
LIN {X 0,Y 554.209,Z 749.56,A -85,B 0,C 180,E1 10253.734,E2 10253.734} C_VEL
LIN {X 0,Y 554.346,Z 749.56,A -85,B 0,C 180,E1 10258.434,E2 10258.434} C_VEL
LIN {X 0,Y 554.261,Z 749.56,A -85,B 0,C 180,E1 10263.122,E2 10263.122} C_VEL
LIN {X 0,Y 554.161,Z 749.56,A -85,B 0,C 180,E1 10267.832,E2 10267.832} C_VEL
LIN {X 0,Y 553.975,Z 749.56,A -85,B 0,C 180,E1 10272.601,E2 10272.601} C_VEL
LIN {X 0,Y 553.891,Z 749.56,A -85,B 0,C 180,E1 10277.46,E2 10277.46} C_VEL
LIN {X 0,Y 553.708,Z 749.56,A -85,B 0,C 180,E1 10282.458,E2 10282.458} C_VEL
LIN {X 0,Y 553.601,Z 749.56,A -85,B 0,C 180,E1 10287.644,E2 10287.644} C_VEL
LIN {X 0,Y 553.428,Z 749.56,A -85,B 0,C 180,E1 10293.095,E2 10293.095} C_VEL
LIN {X 0,Y 553.446,Z 749.56,A -85,B 0,C 180,E1 10296.35,E2 10296.35} C_VEL
LIN {X 0,Y 555.781,Z 755.161,A -85,B 0,C 180,E1 10296.734,E2 10296.734} C_VEL
LIN {X 0,Y 588.144,Z 807.192,A -85,B 0,C 180,E1 10301.112,E2 10301.112} C_VEL
LIN {X 0,Y 603.634,Z 834.721,A -85,B 0,C 180,E1 10303.117,E2 10303.117} C_VEL
LIN {X 0,Y 599.494,Z 886.549,A -85,B 0,C 180,E1 10304.332,E2 10304.332} C_VEL
LIN {X 0,Y 594.53,Z 932.766,A -85,B 0,C 180,E1 10306.002,E2 10306.002} C_VEL
LIN {X 0,Y 587.995,Z 980.571,A -85,B 0,C 180,E1 10308.406,E2 10308.406} C_VEL
LIN {X 0,Y 581.298,Z 1023.202,A -85,B 0,C 180,E1 10311.206,E2 10311.206} C_VEL
LIN {X 0,Y 575.537,Z 1037.455,A -85,B 0,C 180,E1 10312.091,E2 10312.091} C_VEL
LIN {X 0,Y 569.934,Z 1050.86,A -85,B 0,C 180,E1 10313.03,E2 10313.03} C_VEL
LIN {X 0,Y 562.941,Z 1087.421,A -85,B 0,C 180,E1 10316.808,E2 10316.808} C_VEL
LIN {X 0,Y 556.599,Z 1121.966,A -85,B 0,C 180,E1 10321.334,E2 10321.334} C_VEL
LIN {X 0,Y 551.996,Z 1150.341,A -85,B 0,C 180,E1 10326.122,E2 10326.122} C_VEL
LIN {X 0,Y 549.055,Z 1173.426,A -85,B 0,C 180,E1 10331.143,E2 10331.143} C_VEL
LIN {X 0,Y 547.392,Z 1191.152,A -85,B 0,C 180,E1 10336.428,E2 10336.428} C_VEL
LIN {X 0,Y 546.72,Z 1202.219,A -85,B 0,C 180,E1 10341.255,E2 10341.255} C_VEL
LIN {X 0,Y 546.515,Z 1207.659,A -85,B 0,C 180,E1 10345.241,E2 10345.241} C_VEL
LIN {X 0,Y 546.587,Z 1210,A -85,B 0,C 180,E1 10349.999,E2 10349.999} C_VEL
LIN {X 0,Y 546.504,Z 1207.661,A -85,B 0,C 180,E1 10354.757,E2 10354.757} C_VEL
LIN {X 0,Y 546.765,Z 1200.672,A -85,B 0,C 180,E1 10359.544,E2 10359.544} C_VEL
LIN {X 0,Y 547.657,Z 1187.852,A -85,B 0,C 180,E1 10364.73,E2 10364.73} C_VEL
LIN {X 0,Y 549.348,Z 1169.972,A -85,B 0,C 180,E1 10369.689,E2 10369.689} C_VEL
LIN {X 0,Y 552.546,Z 1146.555,A -85,B 0,C 180,E1 10374.601,E2 10374.601} C_VEL
LIN {X 0,Y 557.222,Z 1118.119,A -85,B 0,C 180,E1 10379.218,E2 10379.218} C_VEL
LIN {X 0,Y 563.709,Z 1083.212,A -85,B 0,C 180,E1 10383.691,E2 10383.691} C_VEL
LIN {X 0,Y 570.358,Z 1047.786,A -85,B 0,C 180,E1 10387.241,E2 10387.241} C_VEL
LIN {X 0,Y 577.743,Z 1004.756,A -85,B 0,C 180,E1 10390.546,E2 10390.546} C_VEL
LIN {X 0,Y 584.659,Z 958.639,A -85,B 0,C 180,E1 10393.257,E2 10393.257} C_VEL
LIN {X 0,Y 590.826,Z 910.398,A -85,B 0,C 180,E1 10395.371,E2 10395.371} C_VEL
LIN {X 0,Y 595.881,Z 859.132,A -85,B 0,C 180,E1 10396.881,E2 10396.881} C_VEL
LIN {X 0,Y 597.034,Z 836.677,A -85,B 0,C 180,E1 10397.389,E2 10397.389} C_VEL
LIN {X 0,Y 568.428,Z 785.67,A -85,B 0,C 180,E1 10401.544,E2 10401.544} C_VEL
LIN {X 0,Y 551.342,Z 760.189,A -85,B 0,C 180,E1 10404.383,E2 10404.383} C_VEL
LIN {X 0,Y 548.318,Z 755.636,A -85,B 0,C 180,E1 10404.933,E2 10404.933} C_VEL
LIN {X 0,Y 545.482,Z 750.598,A -85,B 0,C 180,E1 10405.48,E2 10405.48} C_VEL
LIN {X 0,Y 545.423,Z 749.56,A -85,B 0,C 180,E1 10405.592,E2 10405.592} C_VEL
LIN {X 0,Y 545.501,Z 749.56,A -85,B 0,C 180,E1 10411.91,E2 10411.91} C_VEL
LIN {X 0,Y 545.577,Z 749.56,A -85,B 0,C 180,E1 10417.188,E2 10417.188} C_VEL
LIN {X 0,Y 545.842,Z 749.56,A -85,B 0,C 180,E1 10422.274,E2 10422.274} C_VEL
LIN {X 0,Y 546.035,Z 749.56,A -85,B 0,C 180,E1 10427.213,E2 10427.213} C_VEL
LIN {X 0,Y 546.244,Z 749.56,A -85,B 0,C 180,E1 10432.054,E2 10432.054} C_VEL
LIN {X 0,Y 546.354,Z 749.56,A -85,B 0,C 180,E1 10436.833,E2 10436.833} C_VEL
LIN {X 0,Y 546.458,Z 749.56,A -85,B 0,C 180,E1 10441.589,E2 10441.589} C_VEL
LIN {X 0,Y 546.286,Z 749.56,A -85,B 0,C 180,E1 10446.357,E2 10446.357} C_VEL
LIN {X 0,Y 546.055,Z 749.56,A -85,B 0,C 180,E1 10451.174,E2 10451.174} C_VEL
LIN {X 0,Y 545.731,Z 749.56,A -85,B 0,C 180,E1 10456.08,E2 10456.08} C_VEL
LIN {X 0,Y 545.602,Z 749.56,A -85,B 0,C 180,E1 10461.109,E2 10461.109} C_VEL
LIN {X 0,Y 545.458,Z 749.56,A -85,B 0,C 180,E1 10466.318,E2 10466.318} C_VEL
LIN {X 0,Y 545.421,Z 749.568,A -85,B 0,C 180,E1 10470.127,E2 10470.127} C_VEL
LIN {X 0,Y 547.491,Z 754.865,A -85,B 0,C 180,E1 10470.57,E2 10470.57} C_VEL
LIN {X 0,Y 550.309,Z 758.297,A -85,B 0,C 180,E1 10471.076,E2 10471.076} C_VEL
LIN {X 0,Y 570.102,Z 788.034,A -85,B 0,C 180,E1 10474.465,E2 10474.465} C_VEL
LIN {X 0,Y 587.221,Z 820.273,A -85,B 0,C 180,E1 10477.455,E2 10477.455} C_VEL
LIN {X 0,Y 591.232,Z 830.877,A -85,B 0,C 180,E1 10478.267,E2 10478.267} C_VEL
LIN {X 0,Y 586.065,Z 876.308,A -85,B 0,C 180,E1 10479.885,E2 10479.885} C_VEL
LIN {X 0,Y 579.891,Z 918.254,A -85,B 0,C 180,E1 10481.995,E2 10481.995} C_VEL
LIN {X 0,Y 572.737,Z 959.256,A -85,B 0,C 180,E1 10484.762,E2 10484.762} C_VEL
LIN {X 0,Y 565.814,Z 995.516,A -85,B 0,C 180,E1 10487.959,E2 10487.959} C_VEL
LIN {X 0,Y 559.487,Z 1028.691,A -85,B 0,C 180,E1 10491.697,E2 10491.697} C_VEL
LIN {X 0,Y 553.901,Z 1058.994,A -85,B 0,C 180,E1 10496.125,E2 10496.125} C_VEL
LIN {X 0,Y 550.133,Z 1083.245,A -85,B 0,C 180,E1 10500.717,E2 10500.717} C_VEL
LIN {X 0,Y 547.974,Z 1103.264,A -85,B 0,C 180,E1 10505.523,E2 10505.523} C_VEL
LIN {X 0,Y 547.039,Z 1116.389,A -85,B 0,C 180,E1 10509.935,E2 10509.935} C_VEL
LIN {X 0,Y 546.495,Z 1125.814,A -85,B 0,C 180,E1 10514.841,E2 10514.841} C_VEL
LIN {X 0,Y 546.265,Z 1129.478,A -85,B 0,C 180,E1 10518.835,E2 10518.835} C_VEL
LIN {X 0,Y 546.458,Z 1129.104,A -85,B 0,C 180,E1 10523.65,E2 10523.65} C_VEL
LIN {X 0,Y 546.703,Z 1124.97,A -85,B 0,C 180,E1 10527.625,E2 10527.625} C_VEL
LIN {X 0,Y 546.938,Z 1117.327,A -85,B 0,C 180,E1 10531.584,E2 10531.584} C_VEL
LIN {X 0,Y 547.988,Z 1103.447,A -85,B 0,C 180,E1 10536.334,E2 10536.334} C_VEL
LIN {X 0,Y 550.046,Z 1083.687,A -85,B 0,C 180,E1 10541.088,E2 10541.088} C_VEL
LIN {X 0,Y 553.681,Z 1059.816,A -85,B 0,C 180,E1 10545.636,E2 10545.636} C_VEL
LIN {X 0,Y 559.326,Z 1028.914,A -85,B 0,C 180,E1 10550.15,E2 10550.15} C_VEL
LIN {X 0,Y 565.847,Z 994.224,A -85,B 0,C 180,E1 10554.034,E2 10554.034} C_VEL
LIN {X 0,Y 572.673,Z 957.969,A -85,B 0,C 180,E1 10557.185,E2 10557.185} C_VEL
LIN {X 0,Y 579.428,Z 917.857,A -85,B 0,C 180,E1 10559.864,E2 10559.864} C_VEL
LIN {X 0,Y 585.244,Z 876.932,A -85,B 0,C 180,E1 10561.906,E2 10561.906} C_VEL
LIN {X 0,Y 589.911,Z 828.621,A -85,B 0,C 180,E1 10563.651,E2 10563.651} C_VEL
LIN {X 0,Y 572.053,Z 794.01,A -85,B 0,C 180,E1 10566.485,E2 10566.485} C_VEL
LIN {X 0,Y 547.348,Z 754.71,A -85,B 0,C 180,E1 10570.052,E2 10570.052} C_VEL
LIN {X 0,Y 545.445,Z 749.56,A -85,B 0,C 180,E1 10570.415,E2 10570.415} C_VEL
LIN {X 0,Y 545.392,Z 749.56,A -85,B 0,C 180,E1 10576.15,E2 10576.15} C_VEL
LIN {X 0,Y 545.4,Z 749.56,A -85,B 0,C 180,E1 10582.437,E2 10582.437} C_VEL
LIN {X 0,Y 545.372,Z 749.56,A -85,B 0,C 180,E1 10588.228,E2 10588.228} C_VEL
LIN {X 0,Y 545.455,Z 749.56,A -85,B 0,C 180,E1 10593.682,E2 10593.682} C_VEL
LIN {X 0,Y 545.599,Z 749.56,A -85,B 0,C 180,E1 10598.891,E2 10598.891} C_VEL
LIN {X 0,Y 545.72,Z 749.56,A -85,B 0,C 180,E1 10603.919,E2 10603.919} C_VEL
LIN {X 0,Y 546.06,Z 749.56,A -85,B 0,C 180,E1 10608.826,E2 10608.826} C_VEL
LIN {X 0,Y 546.296,Z 749.56,A -85,B 0,C 180,E1 10613.643,E2 10613.643} C_VEL
LIN {X 0,Y 546.444,Z 749.56,A -85,B 0,C 180,E1 10618.411,E2 10618.411} C_VEL
LIN {X 0,Y 546.358,Z 749.56,A -85,B 0,C 180,E1 10623.167,E2 10623.167} C_VEL
LIN {X 0,Y 546.252,Z 749.56,A -85,B 0,C 180,E1 10627.946,E2 10627.946} C_VEL
LIN {X 0,Y 546.05,Z 749.56,A -85,B 0,C 180,E1 10632.787,E2 10632.787} C_VEL
LIN {X 0,Y 545.953,Z 749.56,A -85,B 0,C 180,E1 10637.722,E2 10637.722} C_VEL
LIN {X 0,Y 545.778,Z 749.56,A -85,B 0,C 180,E1 10643.978,E2 10643.978} C_VEL
LIN {X 0,Y 545.581,Z 749.56,A -85,B 0,C 180,E1 10649.9,E2 10649.9} C_VEL
LIN {X 0,Y 545.502,Z 749.56,A -85,B 0,C 180,E1 10655.393,E2 10655.393} C_VEL
LIN {X 0,Y 547.967,Z 755.254,A -85,B 0,C 180,E1 10655.811,E2 10655.811} C_VEL
LIN {X 0,Y 579.897,Z 806.189,A -85,B 0,C 180,E1 10660.272,E2 10660.272} C_VEL
LIN {X 0,Y 597.741,Z 837.781,A -85,B 0,C 180,E1 10662.652,E2 10662.652} C_VEL
LIN {X 0,Y 593.302,Z 889.93,A -85,B 0,C 180,E1 10663.915,E2 10663.915} C_VEL
LIN {X 0,Y 588.146,Z 934.876,A -85,B 0,C 180,E1 10665.596,E2 10665.596} C_VEL
LIN {X 0,Y 581.378,Z 982.003,A -85,B 0,C 180,E1 10668.005,E2 10668.005} C_VEL
LIN {X 0,Y 574.223,Z 1025.237,A -85,B 0,C 180,E1 10670.913,E2 10670.913} C_VEL
LIN {X 0,Y 569.934,Z 1050.86,A -85,B 0,C 180,E1 10673.03,E2 10673.03} C_VEL
LIN {X 0,Y 564.047,Z 1064.086,A -85,B 0,C 180,E1 10674.034,E2 10674.034} C_VEL
LIN {X 0,Y 558.521,Z 1075.172,A -85,B 0,C 180,E1 10674.965,E2 10674.965} C_VEL
LIN {X 0,Y 558.164,Z 1076.664,A -85,B 0,C 180,E1 10675.124,E2 10675.124} C_VEL
LIN {X 0,Y 551.359,Z 1111.176,A -85,B 0,C 180,E1 10679.36,E2 10679.36} C_VEL
LIN {X 0,Y 545.957,Z 1140.942,A -85,B 0,C 180,E1 10684.03,E2 10684.03} C_VEL
LIN {X 0,Y 542.375,Z 1164.737,A -85,B 0,C 180,E1 10688.764,E2 10688.764} C_VEL
LIN {X 0,Y 540.101,Z 1183.698,A -85,B 0,C 180,E1 10693.752,E2 10693.752} C_VEL
LIN {X 0,Y 539.106,Z 1197.612,A -85,B 0,C 180,E1 10698.815,E2 10698.815} C_VEL
LIN {X 0,Y 538.778,Z 1205.908,A -85,B 0,C 180,E1 10703.558,E2 10703.558} C_VEL
LIN {X 0,Y 538.555,Z 1209.666,A -85,B 0,C 180,E1 10708.391,E2 10708.391} C_VEL
LIN {X 0,Y 538.702,Z 1208.902,A -85,B 0,C 180,E1 10713.215,E2 10713.215} C_VEL
LIN {X 0,Y 538.766,Z 1203.543,A -85,B 0,C 180,E1 10718.061,E2 10718.061} C_VEL
LIN {X 0,Y 539.316,Z 1193.42,A -85,B 0,C 180,E1 10722.952,E2 10722.952} C_VEL
LIN {X 0,Y 540.779,Z 1177.999,A -85,B 0,C 180,E1 10727.9,E2 10727.9} C_VEL
LIN {X 0,Y 543.487,Z 1156.98,A -85,B 0,C 180,E1 10732.908,E2 10732.908} C_VEL
LIN {X 0,Y 547.812,Z 1130.454,A -85,B 0,C 180,E1 10737.741,E2 10737.741} C_VEL
LIN {X 0,Y 553.932,Z 1098.043,A -85,B 0,C 180,E1 10742.377,E2 10742.377} C_VEL
LIN {X 0,Y 560.302,Z 1065.013,A -85,B 0,C 180,E1 10746.083,E2 10746.083} C_VEL
LIN {X 0,Y 568.075,Z 1022.052,A -85,B 0,C 180,E1 10749.779,E2 10749.779} C_VEL
LIN {X 0,Y 575.358,Z 978.532,A -85,B 0,C 180,E1 10752.664,E2 10752.664} C_VEL
LIN {X 0,Y 582.318,Z 931.831,A -85,B 0,C 180,E1 10755.015,E2 10755.015} C_VEL
LIN {X 0,Y 587.542,Z 887.642,A -85,B 0,C 180,E1 10756.635,E2 10756.635} C_VEL
LIN {X 0,Y 591.265,Z 839.967,A -85,B 0,C 180,E1 10757.855,E2 10757.855} C_VEL
LIN {X 0,Y 564.173,Z 790.955,A -85,B 0,C 180,E1 10761.976,E2 10761.976} C_VEL
LIN {X 0,Y 545.417,Z 762.474,A -85,B 0,C 180,E1 10765.214,E2 10765.214} C_VEL
LIN {X 0,Y 539.942,Z 755.233,A -85,B 0,C 180,E1 10766.246,E2 10766.246} C_VEL
LIN {X 0,Y 537.543,Z 750.745,A -85,B 0,C 180,E1 10766.747,E2 10766.747} C_VEL
LIN {X 0,Y 537.445,Z 749.56,A -85,B 0,C 180,E1 10766.907,E2 10766.907} C_VEL
LIN {X 0,Y 537.618,Z 749.56,A -85,B 0,C 180,E1 10773.278,E2 10773.278} C_VEL
LIN {X 0,Y 537.725,Z 749.56,A -85,B 0,C 180,E1 10778.576,E2 10778.576} C_VEL
LIN {X 0,Y 537.972,Z 749.56,A -85,B 0,C 180,E1 10783.691,E2 10783.691} C_VEL
LIN {X 0,Y 538.198,Z 749.56,A -85,B 0,C 180,E1 10789.327,E2 10789.327} C_VEL
LIN {X 0,Y 538.503,Z 749.56,A -85,B 0,C 180,E1 10795.175,E2 10795.175} C_VEL
LIN {X 0,Y 538.712,Z 749.56,A -85,B 0,C 180,E1 10800.004,E2 10800.004} C_VEL
LIN {X 0,Y 538.449,Z 749.56,A -85,B 0,C 180,E1 10804.834,E2 10804.834} C_VEL
LIN {X 0,Y 538.15,Z 749.56,A -85,B 0,C 180,E1 10810.646,E2 10810.646} C_VEL
LIN {X 0,Y 537.79,Z 749.56,A -85,B 0,C 180,E1 10816.324,E2 10816.324} C_VEL
LIN {X 0,Y 537.609,Z 749.56,A -85,B 0,C 180,E1 10821.943,E2 10821.943} C_VEL
LIN {X 0,Y 537.557,Z 749.56,A -85,B 0,C 180,E1 10826.735,E2 10826.735} C_VEL
LIN {X 0,Y 537.48,Z 749.56,A -85,B 0,C 180,E1 10828.834,E2 10828.834} C_VEL
LIN {X 0,Y 539.561,Z 754.909,A -85,B 0,C 180,E1 10829.31,E2 10829.31} C_VEL
LIN {X 0,Y 542.579,Z 758.576,A -85,B 0,C 180,E1 10829.886,E2 10829.886} C_VEL
LIN {X 0,Y 562.366,Z 787.55,A -85,B 0,C 180,E1 10833.447,E2 10833.447} C_VEL
LIN {X 0,Y 579.95,Z 819.978,A -85,B 0,C 180,E1 10836.627,E2 10836.627} C_VEL
LIN {X 0,Y 585.472,Z 834.137,A -85,B 0,C 180,E1 10837.784,E2 10837.784} C_VEL
LIN {X 0,Y 579.852,Z 881.241,A -85,B 0,C 180,E1 10839.516,E2 10839.516} C_VEL
LIN {X 0,Y 572.987,Z 924.603,A -85,B 0,C 180,E1 10841.809,E2 10841.809} C_VEL
LIN {X 0,Y 565.852,Z 963.291,A -85,B 0,C 180,E1 10844.518,E2 10844.518} C_VEL
LIN {X 0,Y 558.012,Z 1002.313,A -85,B 0,C 180,E1 10848.115,E2 10848.115} C_VEL
LIN {X 0,Y 551.499,Z 1034.351,A -85,B 0,C 180,E1 10851.94,E2 10851.94} C_VEL
LIN {X 0,Y 545.954,Z 1063.425,A -85,B 0,C 180,E1 10856.388,E2 10856.388} C_VEL
LIN {X 0,Y 541.914,Z 1088.427,A -85,B 0,C 180,E1 10861.451,E2 10861.451} C_VEL
LIN {X 0,Y 539.809,Z 1108.568,A -85,B 0,C 180,E1 10866.927,E2 10866.927} C_VEL
LIN {X 0,Y 538.969,Z 1119.695,A -85,B 0,C 180,E1 10871.191,E2 10871.191} C_VEL
LIN {X 0,Y 538.594,Z 1126.597,A -85,B 0,C 180,E1 10875.375,E2 10875.375} C_VEL
LIN {X 0,Y 538.404,Z 1129.87,A -85,B 0,C 180,E1 10880.306,E2 10880.306} C_VEL
LIN {X 0,Y 538.609,Z 1128.047,A -85,B 0,C 180,E1 10885.173,E2 10885.173} C_VEL
LIN {X 0,Y 538.957,Z 1121.072,A -85,B 0,C 180,E1 10890.001,E2 10890.001} C_VEL
LIN {X 0,Y 539.717,Z 1109.101,A -85,B 0,C 180,E1 10894.819,E2 10894.819} C_VEL
LIN {X 0,Y 541.624,Z 1090.103,A -85,B 0,C 180,E1 10900.043,E2 10900.043} C_VEL
LIN {X 0,Y 545.025,Z 1068.054,A -85,B 0,C 180,E1 10904.656,E2 10904.656} C_VEL
LIN {X 0,Y 550.123,Z 1041.045,A -85,B 0,C 180,E1 10909.015,E2 10909.015} C_VEL
LIN {X 0,Y 556.776,Z 1007.5,A -85,B 0,C 180,E1 10913.176,E2 10913.176} C_VEL
LIN {X 0,Y 563.73,Z 972.239,A -85,B 0,C 180,E1 10916.573,E2 10916.573} C_VEL
LIN {X 0,Y 570.997,Z 932.351,A -85,B 0,C 180,E1 10919.532,E2 10919.532} C_VEL
LIN {X 0,Y 577.616,Z 889.72,A -85,B 0,C 180,E1 10921.88,E2 10921.88} C_VEL
LIN {X 0,Y 583.226,Z 844.377,A -85,B 0,C 180,E1 10923.671,E2 10923.671} C_VEL
LIN {X 0,Y 583.712,Z 831.286,A -85,B 0,C 180,E1 10924.145,E2 10924.145} C_VEL
LIN {X 0,Y 564.781,Z 794.616,A -85,B 0,C 180,E1 10927.242,E2 10927.242} C_VEL
LIN {X 0,Y 539.895,Z 755.17,A -85,B 0,C 180,E1 10930.962,E2 10930.962} C_VEL
LIN {X 0,Y 537.531,Z 749.56,A -85,B 0,C 180,E1 10931.455,E2 10931.455} C_VEL
LIN {X 0,Y 537.384,Z 749.56,A -85,B 0,C 180,E1 10937.548,E2 10937.548} C_VEL
LIN {X 0,Y 537.464,Z 749.56,A -85,B 0,C 180,E1 10943.806,E2 10943.806} C_VEL
LIN {X 0,Y 537.455,Z 749.56,A -85,B 0,C 180,E1 10949.59,E2 10949.59} C_VEL
LIN {X 0,Y 537.562,Z 749.56,A -85,B 0,C 180,E1 10955.055,E2 10955.055} C_VEL
LIN {X 0,Y 537.682,Z 749.56,A -85,B 0,C 180,E1 10960.285,E2 10960.285} C_VEL
LIN {X 0,Y 537.903,Z 749.56,A -85,B 0,C 180,E1 10965.35,E2 10965.35} C_VEL
LIN {X 0,Y 538.255,Z 749.56,A -85,B 0,C 180,E1 10970.298,E2 10970.298} C_VEL
LIN {X 0,Y 538.454,Z 749.56,A -85,B 0,C 180,E1 10975.166,E2 10975.166} C_VEL
LIN {X 0,Y 538.723,Z 749.56,A -85,B 0,C 180,E1 10979.996,E2 10979.996} C_VEL
LIN {X 0,Y 538.424,Z 749.56,A -85,B 0,C 180,E1 10986.441,E2 10986.441} C_VEL
LIN {X 0,Y 538.188,Z 749.56,A -85,B 0,C 180,E1 10991.331,E2 10991.331} C_VEL
LIN {X 0,Y 538.015,Z 749.56,A -85,B 0,C 180,E1 10997.259,E2 10997.259} C_VEL
LIN {X 0,Y 537.844,Z 749.56,A -85,B 0,C 180,E1 11003.159,E2 11003.159} C_VEL
LIN {X 0,Y 537.654,Z 749.56,A -85,B 0,C 180,E1 11009.39,E2 11009.39} C_VEL
LIN {X 0,Y 537.575,Z 749.722,A -85,B 0,C 180,E1 11014.406,E2 11014.406} C_VEL
LIN {X 0,Y 539.891,Z 755.145,A -85,B 0,C 180,E1 11014.814,E2 11014.814} C_VEL
LIN {X 0,Y 567.254,Z 798.124,A -85,B 0,C 180,E1 11018.814,E2 11018.814} C_VEL
LIN {X 0,Y 591.862,Z 841.647,A -85,B 0,C 180,E1 11022.199,E2 11022.199} C_VEL
LIN {X 0,Y 587.371,Z 891.087,A -85,B 0,C 180,E1 11023.424,E2 11023.424} C_VEL
LIN {X 0,Y 581.744,Z 937.148,A -85,B 0,C 180,E1 11025.187,E2 11025.187} C_VEL
LIN {X 0,Y 574.74,Z 983.937,A -85,B 0,C 180,E1 11027.627,E2 11027.627} C_VEL
LIN {X 0,Y 567.233,Z 1026.865,A -85,B 0,C 180,E1 11030.58,E2 11030.58} C_VEL
LIN {X 0,Y 559.934,Z 1067.603,A -85,B 0,C 180,E1 11034.169,E2 11034.169} C_VEL
LIN {X 0,Y 558.164,Z 1076.664,A -85,B 0,C 180,E1 11035.124,E2 11035.124} C_VEL
LIN {X 0,Y 552.294,Z 1088.894,A -85,B 0,C 180,E1 11036.273,E2 11036.273} C_VEL
LIN {X 0,Y 546.75,Z 1099.224,A -85,B 0,C 180,E1 11037.317,E2 11037.317} C_VEL
LIN {X 0,Y 546.392,Z 1100.569,A -85,B 0,C 180,E1 11037.493,E2 11037.493} C_VEL
LIN {X 0,Y 539.954,Z 1133.09,A -85,B 0,C 180,E1 11042.271,E2 11042.271} C_VEL
LIN {X 0,Y 535.577,Z 1158.921,A -85,B 0,C 180,E1 11047.172,E2 11047.172} C_VEL
LIN {X 0,Y 532.884,Z 1179.521,A -85,B 0,C 180,E1 11052.25,E2 11052.25} C_VEL
LIN {X 0,Y 531.512,Z 1193.415,A -85,B 0,C 180,E1 11056.852,E2 11056.852} C_VEL
LIN {X 0,Y 530.896,Z 1203.536,A -85,B 0,C 180,E1 11061.817,E2 11061.817} C_VEL
LIN {X 0,Y 530.754,Z 1208.898,A -85,B 0,C 180,E1 11066.735,E2 11066.735} C_VEL
LIN {X 0,Y 530.939,Z 1209.666,A -85,B 0,C 180,E1 11071.63,E2 11071.63} C_VEL
LIN {X 0,Y 530.854,Z 1205.911,A -85,B 0,C 180,E1 11076.537,E2 11076.537} C_VEL
LIN {X 0,Y 531.227,Z 1197.305,A -85,B 0,C 180,E1 11081.485,E2 11081.485} C_VEL
LIN {X 0,Y 532.316,Z 1183.705,A -85,B 0,C 180,E1 11086.491,E2 11086.491} C_VEL
LIN {X 0,Y 534.733,Z 1164.74,A -85,B 0,C 180,E1 11091.553,E2 11091.553} C_VEL
LIN {X 0,Y 538.888,Z 1139.225,A -85,B 0,C 180,E1 11096.657,E2 11096.657} C_VEL
LIN {X 0,Y 544.763,Z 1108.842,A -85,B 0,C 180,E1 11101.403,E2 11101.403} C_VEL
LIN {X 0,Y 550.872,Z 1077.89,A -85,B 0,C 180,E1 11105.173,E2 11105.173} C_VEL
LIN {X 0,Y 558.657,Z 1037.26,A -85,B 0,C 180,E1 11109.028,E2 11109.028} C_VEL
LIN {X 0,Y 566.284,Z 995.286,A -85,B 0,C 180,E1 11112.114,E2 11112.114} C_VEL
LIN {X 0,Y 573.486,Z 950.851,A -85,B 0,C 180,E1 11114.652,E2 11114.652} C_VEL
LIN {X 0,Y 579.75,Z 904.576,A -85,B 0,C 180,E1 11116.612,E2 11116.612} C_VEL
LIN {X 0,Y 585.033,Z 854.063,A -85,B 0,C 180,E1 11118.082,E2 11118.082} C_VEL
LIN {X 0,Y 585.461,Z 843.267,A -85,B 0,C 180,E1 11118.347,E2 11118.347} C_VEL
LIN {X 0,Y 560.113,Z 796.454,A -85,B 0,C 180,E1 11122.389,E2 11122.389} C_VEL
LIN {X 0,Y 542.104,Z 768.9,A -85,B 0,C 180,E1 11125.578,E2 11125.578} C_VEL
LIN {X 0,Y 532.674,Z 755.853,A -85,B 0,C 180,E1 11127.444,E2 11127.444} C_VEL
LIN {X 0,Y 529.728,Z 751.274,A -85,B 0,C 180,E1 11128.077,E2 11128.077} C_VEL
LIN {X 0,Y 529.503,Z 749.56,A -85,B 0,C 180,E1 11128.284,E2 11128.284} C_VEL
LIN {X 0,Y 529.648,Z 749.56,A -85,B 0,C 180,E1 11132.843,E2 11132.843} C_VEL
LIN {X 0,Y 529.794,Z 749.56,A -85,B 0,C 180,E1 11138.239,E2 11138.239} C_VEL
LIN {X 0,Y 530.059,Z 749.56,A -85,B 0,C 180,E1 11143.44,E2 11143.44} C_VEL
LIN {X 0,Y 530.25,Z 749.56,A -85,B 0,C 180,E1 11148.497,E2 11148.497} C_VEL
LIN {X 0,Y 530.518,Z 749.56,A -85,B 0,C 180,E1 11153.462,E2 11153.462} C_VEL
LIN {X 0,Y 530.81,Z 749.56,A -85,B 0,C 180,E1 11160.005,E2 11160.005} C_VEL
LIN {X 0,Y 530.557,Z 749.56,A -85,B 0,C 180,E1 11164.906,E2 11164.906} C_VEL
LIN {X 0,Y 530.342,Z 749.56,A -85,B 0,C 180,E1 11169.848,E2 11169.848} C_VEL
LIN {X 0,Y 529.982,Z 749.56,A -85,B 0,C 180,E1 11174.874,E2 11174.874} C_VEL
LIN {X 0,Y 529.776,Z 749.56,A -85,B 0,C 180,E1 11180.022,E2 11180.022} C_VEL
LIN {X 0,Y 529.645,Z 749.56,A -85,B 0,C 180,E1 11185.344,E2 11185.344} C_VEL
LIN {X 0,Y 529.624,Z 750.316,A -85,B 0,C 180,E1 11187.484,E2 11187.484} C_VEL
LIN {X 0,Y 532.161,Z 755.416,A -85,B 0,C 180,E1 11188.066,E2 11188.066} C_VEL
LIN {X 0,Y 534.763,Z 758.634,A -85,B 0,C 180,E1 11188.596,E2 11188.596} C_VEL
LIN {X 0,Y 552.933,Z 784.834,A -85,B 0,C 180,E1 11192.071,E2 11192.071} C_VEL
LIN {X 0,Y 570.387,Z 814.91,A -85,B 0,C 180,E1 11195.296,E2 11195.296} C_VEL
LIN {X 0,Y 579.858,Z 837.066,A -85,B 0,C 180,E1 11197.284,E2 11197.284} C_VEL
LIN {X 0,Y 574.148,Z 882.765,A -85,B 0,C 180,E1 11198.997,E2 11198.997} C_VEL
LIN {X 0,Y 566.799,Z 927.13,A -85,B 0,C 180,E1 11201.384,E2 11201.384} C_VEL
LIN {X 0,Y 559.173,Z 966.104,A -85,B 0,C 180,E1 11204.179,E2 11204.179} C_VEL
LIN {X 0,Y 551.143,Z 1004.233,A -85,B 0,C 180,E1 11207.764,E2 11207.764} C_VEL
LIN {X 0,Y 543.897,Z 1038.065,A -85,B 0,C 180,E1 11211.924,E2 11211.924} C_VEL
LIN {X 0,Y 538.296,Z 1065.829,A -85,B 0,C 180,E1 11216.33,E2 11216.33} C_VEL
LIN {X 0,Y 534.275,Z 1089.624,A -85,B 0,C 180,E1 11221.27,E2 11221.27} C_VEL
LIN {X 0,Y 531.988,Z 1108.153,A -85,B 0,C 180,E1 11226.568,E2 11226.568} C_VEL
LIN {X 0,Y 531.126,Z 1119.403,A -85,B 0,C 180,E1 11230.902,E2 11230.902} C_VEL
LIN {X 0,Y 530.658,Z 1126.853,A -85,B 0,C 180,E1 11235.535,E2 11235.535} C_VEL
LIN {X 0,Y 530.496,Z 1129.841,A -85,B 0,C 180,E1 11240.16,E2 11240.16} C_VEL
LIN {X 0,Y 530.722,Z 1128.188,A -85,B 0,C 180,E1 11245.101,E2 11245.101} C_VEL
LIN {X 0,Y 530.987,Z 1122.878,A -85,B 0,C 180,E1 11249.186,E2 11249.186} C_VEL
LIN {X 0,Y 531.788,Z 1111.777,A -85,B 0,C 180,E1 11254.075,E2 11254.075} C_VEL
LIN {X 0,Y 533.584,Z 1094.497,A -85,B 0,C 180,E1 11259.373,E2 11259.373} C_VEL
LIN {X 0,Y 537.136,Z 1071.877,A -85,B 0,C 180,E1 11264.428,E2 11264.428} C_VEL
LIN {X 0,Y 542.892,Z 1042.365,A -85,B 0,C 180,E1 11269.33,E2 11269.33} C_VEL
LIN {X 0,Y 549.763,Z 1009.473,A -85,B 0,C 180,E1 11273.489,E2 11273.489} C_VEL
LIN {X 0,Y 556.969,Z 974.578,A -85,B 0,C 180,E1 11276.921,E2 11276.921} C_VEL
LIN {X 0,Y 564.728,Z 933.528,A -85,B 0,C 180,E1 11280.004,E2 11280.004} C_VEL
LIN {X 0,Y 571.473,Z 891.858,A -85,B 0,C 180,E1 11282.331,E2 11282.331} C_VEL
LIN {X 0,Y 577.328,Z 846.702,A -85,B 0,C 180,E1 11284.15,E2 11284.15} C_VEL
LIN {X 0,Y 577.838,Z 834.574,A -85,B 0,C 180,E1 11284.589,E2 11284.589} C_VEL
LIN {X 0,Y 557.805,Z 795.817,A -85,B 0,C 180,E1 11287.977,E2 11287.977} C_VEL
LIN {X 0,Y 532.376,Z 755.596,A -85,B 0,C 180,E1 11291.92,E2 11291.92} C_VEL
LIN {X 0,Y 529.583,Z 750.387,A -85,B 0,C 180,E1 11292.4,E2 11292.4} C_VEL
LIN {X 0,Y 529.53,Z 749.56,A -85,B 0,C 180,E1 11293.228,E2 11293.228} C_VEL
LIN {X 0,Y 529.473,Z 749.56,A -85,B 0,C 180,E1 11298.965,E2 11298.965} C_VEL
LIN {X 0,Y 529.517,Z 749.56,A -85,B 0,C 180,E1 11305.191,E2 11305.191} C_VEL
LIN {X 0,Y 529.572,Z 749.56,A -85,B 0,C 180,E1 11310.976,E2 11310.976} C_VEL
LIN {X 0,Y 529.664,Z 749.56,A -85,B 0,C 180,E1 11316.453,E2 11316.453} C_VEL
LIN {X 0,Y 529.798,Z 749.56,A -85,B 0,C 180,E1 11321.709,E2 11321.709} C_VEL
LIN {X 0,Y 530.085,Z 749.56,A -85,B 0,C 180,E1 11326.812,E2 11326.812} C_VEL
LIN {X 0,Y 530.426,Z 749.56,A -85,B 0,C 180,E1 11331.806,E2 11331.806} C_VEL
LIN {X 0,Y 530.667,Z 749.56,A -85,B 0,C 180,E1 11336.731,E2 11336.731} C_VEL
LIN {X 0,Y 530.742,Z 749.56,A -85,B 0,C 180,E1 11341.627,E2 11341.627} C_VEL
LIN {X 0,Y 530.515,Z 749.56,A -85,B 0,C 180,E1 11346.538,E2 11346.538} C_VEL
LIN {X 0,Y 530.262,Z 749.56,A -85,B 0,C 180,E1 11351.502,E2 11351.502} C_VEL
LIN {X 0,Y 530.154,Z 749.56,A -85,B 0,C 180,E1 11356.557,E2 11356.557} C_VEL
LIN {X 0,Y 529.948,Z 749.56,A -85,B 0,C 180,E1 11361.754,E2 11361.754} C_VEL
LIN {X 0,Y 529.769,Z 749.56,A -85,B 0,C 180,E1 11367.839,E2 11367.839} C_VEL
LIN {X 0,Y 529.608,Z 749.767,A -85,B 0,C 180,E1 11373.361,E2 11373.361} C_VEL
LIN {X 0,Y 531.915,Z 755.133,A -85,B 0,C 180,E1 11373.783,E2 11373.783} C_VEL
LIN {X 0,Y 555.184,Z 790.916,A -85,B 0,C 180,E1 11377.348,E2 11377.348} C_VEL
LIN {X 0,Y 582.111,Z 837.172,A -85,B 0,C 180,E1 11381.142,E2 11381.142} C_VEL
LIN {X 0,Y 585.997,Z 844.415,A -85,B 0,C 180,E1 11381.711,E2 11381.711} C_VEL
LIN {X 0,Y 581.292,Z 893.372,A -85,B 0,C 180,E1 11382.963,E2 11382.963} C_VEL
LIN {X 0,Y 575.201,Z 940.533,A -85,B 0,C 180,E1 11384.819,E2 11384.819} C_VEL
LIN {X 0,Y 568.129,Z 985.645,A -85,B 0,C 180,E1 11387.227,E2 11387.227} C_VEL
LIN {X 0,Y 560.078,Z 1029.699,A -85,B 0,C 180,E1 11390.34,E2 11390.34} C_VEL
LIN {X 0,Y 552.552,Z 1069.621,A -85,B 0,C 180,E1 11393.949,E2 11393.949} C_VEL
LIN {X 0,Y 546.392,Z 1100.569,A -85,B 0,C 180,E1 11397.493,E2 11397.493} C_VEL
LIN {X 0,Y 540.501,Z 1111.806,A -85,B 0,C 180,E1 11398.777,E2 11398.777} C_VEL
LIN {X 0,Y 535.077,Z 1121.233,A -85,B 0,C 180,E1 11399.938,E2 11399.938} C_VEL
LIN {X 0,Y 534.763,Z 1122.469,A -85,B 0,C 180,E1 11400.129,E2 11400.129} C_VEL
LIN {X 0,Y 529.386,Z 1150.531,A -85,B 0,C 180,E1 11405.075,E2 11405.075} C_VEL
LIN {X 0,Y 525.853,Z 1173.388,A -85,B 0,C 180,E1 11410.265,E2 11410.265} C_VEL
LIN {X 0,Y 523.977,Z 1189.997,A -85,B 0,C 180,E1 11415.383,E2 11415.383} C_VEL
LIN {X 0,Y 523.165,Z 1200.66,A -85,B 0,C 180,E1 11420.019,E2 11420.019} C_VEL
LIN {X 0,Y 522.821,Z 1207.65,A -85,B 0,C 180,E1 11425.025,E2 11425.025} C_VEL
LIN {X 0,Y 522.91,Z 1210,A -85,B 0,C 180,E1 11429.999,E2 11429.999} C_VEL
LIN {X 0,Y 522.816,Z 1207.653,A -85,B 0,C 180,E1 11434.974,E2 11434.974} C_VEL
LIN {X 0,Y 523.13,Z 1200.663,A -85,B 0,C 180,E1 11439.98,E2 11439.98} C_VEL
LIN {X 0,Y 524.153,Z 1188.208,A -85,B 0,C 180,E1 11445.28,E2 11445.28} C_VEL
LIN {X 0,Y 526.192,Z 1170.561,A -85,B 0,C 180,E1 11450.444,E2 11450.444} C_VEL
LIN {X 0,Y 529.879,Z 1147.271,A -85,B 0,C 180,E1 11455.579,E2 11455.579} C_VEL
LIN {X 0,Y 535.406,Z 1119.568,A -85,B 0,C 180,E1 11460.297,E2 11460.297} C_VEL
LIN {X 0,Y 540.941,Z 1092.151,A -85,B 0,C 180,E1 11463.965,E2 11463.965} C_VEL
LIN {X 0,Y 548.7,Z 1053.337,A -85,B 0,C 180,E1 11468.062,E2 11468.062} C_VEL
LIN {X 0,Y 556.795,Z 1011.864,A -85,B 0,C 180,E1 11471.464,E2 11471.464} C_VEL
LIN {X 0,Y 564.779,Z 966.287,A -85,B 0,C 180,E1 11474.381,E2 11474.381} C_VEL
LIN {X 0,Y 572.368,Z 915.991,A -85,B 0,C 180,E1 11476.742,E2 11476.742} C_VEL
LIN {X 0,Y 578.142,Z 868.882,A -85,B 0,C 180,E1 11478.28,E2 11478.28} C_VEL
LIN {X 0,Y 579.819,Z 846.796,A -85,B 0,C 180,E1 11478.838,E2 11478.838} C_VEL
LIN {X 0,Y 556.157,Z 802.015,A -85,B 0,C 180,E1 11482.801,E2 11482.801} C_VEL
LIN {X 0,Y 538.585,Z 775.004,A -85,B 0,C 180,E1 11485.991,E2 11485.991} C_VEL
LIN {X 0,Y 528.599,Z 761.41,A -85,B 0,C 180,E1 11488.015,E2 11488.015} C_VEL
LIN {X 0,Y 525.05,Z 756.078,A -85,B 0,C 180,E1 11488.803,E2 11488.803} C_VEL
LIN {X 0,Y 521.745,Z 751.072,A -85,B 0,C 180,E1 11489.565,E2 11489.565} C_VEL
LIN {X 0,Y 521.594,Z 749.56,A -85,B 0,C 180,E1 11489.728,E2 11489.728} C_VEL
LIN {X 0,Y 521.736,Z 749.56,A -85,B 0,C 180,E1 11494.254,E2 11494.254} C_VEL
LIN {X 0,Y 521.953,Z 749.56,A -85,B 0,C 180,E1 11499.675,E2 11499.675} C_VEL
LIN {X 0,Y 522.195,Z 749.56,A -85,B 0,C 180,E1 11504.908,E2 11504.908} C_VEL
LIN {X 0,Y 522.427,Z 749.56,A -85,B 0,C 180,E1 11510.01,E2 11510.01} C_VEL
LIN {X 0,Y 522.694,Z 749.56,A -85,B 0,C 180,E1 11515.029,E2 11515.029} C_VEL
LIN {X 0,Y 522.911,Z 749.56,A -85,B 0,C 180,E1 11520.005,E2 11520.005} C_VEL
LIN {X 0,Y 522.644,Z 749.56,A -85,B 0,C 180,E1 11524.981,E2 11524.981} C_VEL
LIN {X 0,Y 522.377,Z 749.56,A -85,B 0,C 180,E1 11530.412,E2 11530.412} C_VEL
LIN {X 0,Y 522.039,Z 749.56,A -85,B 0,C 180,E1 11535.106,E2 11535.106} C_VEL
LIN {X 0,Y 521.831,Z 749.56,A -85,B 0,C 180,E1 11540.34,E2 11540.34} C_VEL
LIN {X 0,Y 521.668,Z 749.561,A -85,B 0,C 180,E1 11545.967,E2 11545.967} C_VEL
LIN {X 0,Y 523.567,Z 754.67,A -85,B 0,C 180,E1 11546.473,E2 11546.473} C_VEL
LIN {X 0,Y 526.81,Z 758.338,A -85,B 0,C 180,E1 11547.178,E2 11547.178} C_VEL
LIN {X 0,Y 545.101,Z 784.38,A -85,B 0,C 180,E1 11550.898,E2 11550.898} C_VEL
LIN {X 0,Y 562.706,Z 813.809,A -85,B 0,C 180,E1 11554.277,E2 11554.277} C_VEL
LIN {X 0,Y 574.264,Z 840.208,A -85,B 0,C 180,E1 11556.779,E2 11556.779} C_VEL
LIN {X 0,Y 568.224,Z 885.8,A -85,B 0,C 180,E1 11558.54,E2 11558.54} C_VEL
LIN {X 0,Y 560.521,Z 930.313,A -85,B 0,C 180,E1 11560.988,E2 11560.988} C_VEL
LIN {X 0,Y 552.549,Z 968.826,A -85,B 0,C 180,E1 11563.823,E2 11563.823} C_VEL
LIN {X 0,Y 544.468,Z 1005.506,A -85,B 0,C 180,E1 11567.335,E2 11567.335} C_VEL
LIN {X 0,Y 536.828,Z 1039.27,A -85,B 0,C 180,E1 11571.558,E2 11571.558} C_VEL
LIN {X 0,Y 531.039,Z 1066.511,A -85,B 0,C 180,E1 11575.951,E2 11575.951} C_VEL
LIN {X 0,Y 526.793,Z 1089.695,A -85,B 0,C 180,E1 11580.815,E2 11580.815} C_VEL
LIN {X 0,Y 524.448,Z 1106.587,A -85,B 0,C 180,E1 11585.604,E2 11585.604} C_VEL
LIN {X 0,Y 523.27,Z 1119.128,A -85,B 0,C 180,E1 11590.604,E2 11590.604} C_VEL
LIN {X 0,Y 522.811,Z 1126.305,A -85,B 0,C 180,E1 11594.923,E2 11594.923} C_VEL
LIN {X 0,Y 522.571,Z 1129.812,A -85,B 0,C 180,E1 11600.009,E2 11600.009} C_VEL
LIN {X 0,Y 522.808,Z 1128.319,A -85,B 0,C 180,E1 11605.026,E2 11605.026} C_VEL
LIN {X 0,Y 523.084,Z 1123.135,A -85,B 0,C 180,E1 11609.173,E2 11609.173} C_VEL
LIN {X 0,Y 524.033,Z 1111.513,A -85,B 0,C 180,E1 11614.549,E2 11614.549} C_VEL
LIN {X 0,Y 525.885,Z 1095.717,A -85,B 0,C 180,E1 11619.511,E2 11619.511} C_VEL
LIN {X 0,Y 529.64,Z 1073.116,A -85,B 0,C 180,E1 11624.676,E2 11624.676} C_VEL
LIN {X 0,Y 535.467,Z 1044.66,A -85,B 0,C 180,E1 11629.505,E2 11629.505} C_VEL
LIN {X 0,Y 542.361,Z 1013.183,A -85,B 0,C 180,E1 11633.611,E2 11633.611} C_VEL
LIN {X 0,Y 550.245,Z 976.838,A -85,B 0,C 180,E1 11637.277,E2 11637.277} C_VEL
LIN {X 0,Y 558.213,Z 936.083,A -85,B 0,C 180,E1 11640.39,E2 11640.39} C_VEL
LIN {X 0,Y 564.975,Z 896.304,A -85,B 0,C 180,E1 11642.681,E2 11642.681} C_VEL
LIN {X 0,Y 571.429,Z 848.762,A -85,B 0,C 180,E1 11644.643,E2 11644.643} C_VEL
LIN {X 0,Y 571.833,Z 837.719,A -85,B 0,C 180,E1 11645.065,E2 11645.065} C_VEL
LIN {X 0,Y 552.199,Z 799.484,A -85,B 0,C 180,E1 11648.503,E2 11648.503} C_VEL
LIN {X 0,Y 528.948,Z 762.132,A -85,B 0,C 180,E1 11652.238,E2 11652.238} C_VEL
LIN {X 0,Y 521.815,Z 751.278,A -85,B 0,C 180,E1 11653.449,E2 11653.449} C_VEL
LIN {X 0,Y 521.618,Z 749.56,A -85,B 0,C 180,E1 11653.585,E2 11653.585} C_VEL
LIN {X 0,Y 521.583,Z 749.56,A -85,B 0,C 180,E1 11658.876,E2 11658.876} C_VEL
LIN {X 0,Y 521.543,Z 749.56,A -85,B 0,C 180,E1 11664.579,E2 11664.579} C_VEL
LIN {X 0,Y 521.596,Z 749.56,A -85,B 0,C 180,E1 11670.488,E2 11670.488} C_VEL
LIN {X 0,Y 521.747,Z 749.56,A -85,B 0,C 180,E1 11676.073,E2 11676.073} C_VEL
LIN {X 0,Y 521.868,Z 749.56,A -85,B 0,C 180,E1 11681.421,E2 11681.421} C_VEL
LIN {X 0,Y 522.159,Z 749.56,A -85,B 0,C 180,E1 11686.608,E2 11686.608} C_VEL
LIN {X 0,Y 522.504,Z 749.56,A -85,B 0,C 180,E1 11691.681,E2 11691.681} C_VEL
LIN {X 0,Y 522.776,Z 749.56,A -85,B 0,C 180,E1 11696.681,E2 11696.681} C_VEL
LIN {X 0,Y 522.849,Z 749.56,A -85,B 0,C 180,E1 11701.652,E2 11701.652} C_VEL
LIN {X 0,Y 522.596,Z 749.56,A -85,B 0,C 180,E1 11706.637,E2 11706.637} C_VEL
LIN {X 0,Y 522.354,Z 749.56,A -85,B 0,C 180,E1 11711.679,E2 11711.679} C_VEL
LIN {X 0,Y 522.175,Z 749.56,A -85,B 0,C 180,E1 11717.253,E2 11717.253} C_VEL
LIN {X 0,Y 522.006,Z 749.56,A -85,B 0,C 180,E1 11722.125,E2 11722.125} C_VEL
LIN {X 0,Y 521.893,Z 749.56,A -85,B 0,C 180,E1 11727.594,E2 11727.594} C_VEL
LIN {X 0,Y 521.712,Z 750.167,A -85,B 0,C 180,E1 11732.281,E2 11732.281} C_VEL
LIN {X 0,Y 524.487,Z 755.567,A -85,B 0,C 180,E1 11732.787,E2 11732.787} C_VEL
LIN {X 0,Y 548.232,Z 792.304,A -85,B 0,C 180,E1 11736.571,E2 11736.571} C_VEL
LIN {X 0,Y 572.845,Z 834.292,A -85,B 0,C 180,E1 11740.14,E2 11740.14} C_VEL
LIN {X 0,Y 580.067,Z 847.609,A -85,B 0,C 180,E1 11741.221,E2 11741.221} C_VEL
LIN {X 0,Y 575.16,Z 895.85,A -85,B 0,C 180,E1 11742.507,E2 11742.507} C_VEL
LIN {X 0,Y 568.631,Z 944.544,A -85,B 0,C 180,E1 11744.477,E2 11744.477} C_VEL
LIN {X 0,Y 561.201,Z 989.063,A -85,B 0,C 180,E1 11746.943,E2 11746.943} C_VEL
LIN {X 0,Y 552.663,Z 1033.852,A -85,B 0,C 180,E1 11750.198,E2 11750.198} C_VEL
LIN {X 0,Y 544.9,Z 1072.755,A -85,B 0,C 180,E1 11753.854,E2 11753.854} C_VEL
LIN {X 0,Y 537.946,Z 1107.653,A -85,B 0,C 180,E1 11757.979,E2 11757.979} C_VEL
LIN {X 0,Y 534.763,Z 1122.469,A -85,B 0,C 180,E1 11760.129,E2 11760.129} C_VEL
LIN {X 0,Y 529.172,Z 1132.54,A -85,B 0,C 180,E1 11761.56,E2 11761.56} C_VEL
LIN {X 0,Y 523.641,Z 1142.016,A -85,B 0,C 180,E1 11763.043,E2 11763.043} C_VEL
LIN {X 0,Y 519.301,Z 1165.823,A -85,B 0,C 180,E1 11768.048,E2 11768.048} C_VEL
LIN {X 0,Y 516.598,Z 1185.03,A -85,B 0,C 180,E1 11773.428,E2 11773.428} C_VEL
LIN {X 0,Y 515.478,Z 1197.296,A -85,B 0,C 180,E1 11778.158,E2 11778.158} C_VEL
LIN {X 0,Y 515.095,Z 1205.908,A -85,B 0,C 180,E1 11783.26,E2 11783.26} C_VEL
LIN {X 0,Y 514.869,Z 1209.666,A -85,B 0,C 180,E1 11788.317,E2 11788.317} C_VEL
LIN {X 0,Y 515.131,Z 1209.666,A -85,B 0,C 180,E1 11791.68,E2 11791.68} C_VEL
LIN {X 0,Y 515.075,Z 1205.911,A -85,B 0,C 180,E1 11796.738,E2 11796.738} C_VEL
LIN {X 0,Y 515.472,Z 1197.299,A -85,B 0,C 180,E1 11801.841,E2 11801.841} C_VEL
LIN {X 0,Y 516.761,Z 1183.703,A -85,B 0,C 180,E1 11807.002,E2 11807.002} C_VEL
LIN {X 0,Y 519.49,Z 1164.741,A -85,B 0,C 180,E1 11812.218,E2 11812.218} C_VEL
LIN {X 0,Y 524.187,Z 1139.221,A -85,B 0,C 180,E1 11817.467,E2 11817.467} C_VEL
LIN {X 0,Y 529.141,Z 1114.769,A -85,B 0,C 180,E1 11821.411,E2 11821.411} C_VEL
LIN {X 0,Y 536.181,Z 1080.605,A -85,B 0,C 180,E1 11825.711,E2 11825.711} C_VEL
LIN {X 0,Y 544.72,Z 1039.295,A -85,B 0,C 180,E1 11829.778,E2 11829.778} C_VEL
LIN {X 0,Y 552.993,Z 998.074,A -85,B 0,C 180,E1 11832.932,E2 11832.932} C_VEL
LIN {X 0,Y 561.022,Z 953.074,A -85,B 0,C 180,E1 11835.601,E2 11835.601} C_VEL
LIN {X 0,Y 568.097,Z 906.65,A -85,B 0,C 180,E1 11837.652,E2 11837.652} C_VEL
LIN {X 0,Y 573.968,Z 855.737,A -85,B 0,C 180,E1 11839.185,E2 11839.185} C_VEL
LIN {X 0,Y 573.956,Z 849.815,A -85,B 0,C 180,E1 11839.39,E2 11839.39} C_VEL
LIN {X 0,Y 552.224,Z 807.525,A -85,B 0,C 180,E1 11843.221,E2 11843.221} C_VEL
LIN {X 0,Y 534.876,Z 780.717,A -85,B 0,C 180,E1 11846.454,E2 11846.454} C_VEL
LIN {X 0,Y 521.54,Z 762.28,A -85,B 0,C 180,E1 11849.296,E2 11849.296} C_VEL
LIN {X 0,Y 517.337,Z 756.183,A -85,B 0,C 180,E1 11850.292,E2 11850.292} C_VEL
LIN {X 0,Y 514.012,Z 751.661,A -85,B 0,C 180,E1 11851.108,E2 11851.108} C_VEL
LIN {X 0,Y 513.749,Z 749.56,A -85,B 0,C 180,E1 11851.332,E2 11851.332} C_VEL
LIN {X 0,Y 513.883,Z 749.56,A -85,B 0,C 180,E1 11857.53,E2 11857.53} C_VEL
LIN {X 0,Y 514.193,Z 749.56,A -85,B 0,C 180,E1 11862.914,E2 11862.914} C_VEL
LIN {X 0,Y 514.41,Z 749.56,A -85,B 0,C 180,E1 11868.138,E2 11868.138} C_VEL
LIN {X 0,Y 514.705,Z 749.56,A -85,B 0,C 180,E1 11873.26,E2 11873.26} C_VEL
LIN {X 0,Y 514.927,Z 749.56,A -85,B 0,C 180,E1 11878.323,E2 11878.323} C_VEL
LIN {X 0,Y 514.828,Z 749.56,A -85,B 0,C 180,E1 11883.664,E2 11883.664} C_VEL
LIN {X 0,Y 514.604,Z 749.56,A -85,B 0,C 180,E1 11888.448,E2 11888.448} C_VEL
LIN {X 0,Y 514.171,Z 749.56,A -85,B 0,C 180,E1 11894.107,E2 11894.107} C_VEL
LIN {X 0,Y 513.908,Z 749.56,A -85,B 0,C 180,E1 11900.668,E2 11900.668} C_VEL
LIN {X 0,Y 513.81,Z 750.131,A -85,B 0,C 180,E1 11904.378,E2 11904.378} C_VEL
LIN {X 0,Y 516.125,Z 755.21,A -85,B 0,C 180,E1 11905.011,E2 11905.011} C_VEL
LIN {X 0,Y 518.971,Z 758.182,A -85,B 0,C 180,E1 11905.672,E2 11905.672} C_VEL
LIN {X 0,Y 537.552,Z 784.365,A -85,B 0,C 180,E1 11909.706,E2 11909.706} C_VEL
LIN {X 0,Y 555.051,Z 813.173,A -85,B 0,C 180,E1 11913.229,E2 11913.229} C_VEL
LIN {X 0,Y 568.786,Z 843.104,A -85,B 0,C 180,E1 11916.26,E2 11916.26} C_VEL
LIN {X 0,Y 562.638,Z 887.104,A -85,B 0,C 180,E1 11917.99,E2 11917.99} C_VEL
LIN {X 0,Y 554.698,Z 931.263,A -85,B 0,C 180,E1 11920.441,E2 11920.441} C_VEL
LIN {X 0,Y 546.505,Z 969.189,A -85,B 0,C 180,E1 11923.254,E2 11923.254} C_VEL
LIN {X 0,Y 538.062,Z 1005.635,A -85,B 0,C 180,E1 11926.766,E2 11926.766} C_VEL
LIN {X 0,Y 530.249,Z 1038.463,A -85,B 0,C 180,E1 11930.892,E2 11930.892} C_VEL
LIN {X 0,Y 524.077,Z 1066.049,A -85,B 0,C 180,E1 11935.343,E2 11935.343} C_VEL
LIN {X 0,Y 519.378,Z 1089.785,A -85,B 0,C 180,E1 11940.357,E2 11940.357} C_VEL
LIN {X 0,Y 516.716,Z 1107.461,A -85,B 0,C 180,E1 11945.424,E2 11945.424} C_VEL
LIN {X 0,Y 515.446,Z 1119.82,A -85,B 0,C 180,E1 11950.455,E2 11950.455} C_VEL
LIN {X 0,Y 514.8,Z 1127.355,A -85,B 0,C 180,E1 11955.644,E2 11955.644} C_VEL
LIN {X 0,Y 514.656,Z 1129.858,A -85,B 0,C 180,E1 11959.854,E2 11959.854} C_VEL
LIN {X 0,Y 514.905,Z 1128.538,A -85,B 0,C 180,E1 11964.95,E2 11964.95} C_VEL
LIN {X 0,Y 515.214,Z 1123.793,A -85,B 0,C 180,E1 11969.161,E2 11969.161} C_VEL
LIN {X 0,Y 516.224,Z 1112.528,A -85,B 0,C 180,E1 11974.618,E2 11974.618} C_VEL
LIN {X 0,Y 518.187,Z 1096.937,A -85,B 0,C 180,E1 11979.654,E2 11979.654} C_VEL
LIN {X 0,Y 522.112,Z 1074.535,A -85,B 0,C 180,E1 11984.885,E2 11984.885} C_VEL
LIN {X 0,Y 528.019,Z 1047.1,A -85,B 0,C 180,E1 11989.661,E2 11989.661} C_VEL
LIN {X 0,Y 534.956,Z 1016.85,A -85,B 0,C 180,E1 11993.737,E2 11993.737} C_VEL
LIN {X 0,Y 543.221,Z 980.052,A -85,B 0,C 180,E1 11997.547,E2 11997.547} C_VEL
LIN {X 0,Y 551.111,Z 941.443,A -85,B 0,C 180,E1 12000.597,E2 12000.597} C_VEL
LIN {X 0,Y 558.62,Z 900.068,A -85,B 0,C 180,E1 12003.065,E2 12003.065} C_VEL
LIN {X 0,Y 565.067,Z 854.769,A -85,B 0,C 180,E1 12004.999,E2 12004.999} C_VEL
LIN {X 0,Y 565.958,Z 841.102,A -85,B 0,C 180,E1 12005.526,E2 12005.526} C_VEL
LIN {X 0,Y 545.684,Z 801.308,A -85,B 0,C 180,E1 12009.209,E2 12009.209} C_VEL
LIN {X 0,Y 521.148,Z 762.186,A -85,B 0,C 180,E1 12013.304,E2 12013.304} C_VEL
LIN {X 0,Y 513.865,Z 751.263,A -85,B 0,C 180,E1 12014.6,E2 12014.6} C_VEL
LIN {X 0,Y 513.653,Z 749.56,A -85,B 0,C 180,E1 12014.747,E2 12014.747} C_VEL
LIN {X 0,Y 513.657,Z 749.56,A -85,B 0,C 180,E1 12019.899,E2 12019.899} C_VEL
LIN {X 0,Y 513.596,Z 749.56,A -85,B 0,C 180,E1 12026.005,E2 12026.005} C_VEL
LIN {X 0,Y 513.714,Z 749.56,A -85,B 0,C 180,E1 12031.944,E2 12031.944} C_VEL
LIN {X 0,Y 513.849,Z 749.56,A -85,B 0,C 180,E1 12037.518,E2 12037.518} C_VEL
LIN {X 0,Y 514.01,Z 749.56,A -85,B 0,C 180,E1 12042.898,E2 12042.898} C_VEL
LIN {X 0,Y 514.366,Z 749.56,A -85,B 0,C 180,E1 12048.127,E2 12048.127} C_VEL
LIN {X 0,Y 514.664,Z 749.56,A -85,B 0,C 180,E1 12053.25,E2 12053.25} C_VEL
LIN {X 0,Y 514.853,Z 749.56,A -85,B 0,C 180,E1 12058.313,E2 12058.313} C_VEL
LIN {X 0,Y 514.755,Z 749.56,A -85,B 0,C 180,E1 12063.508,E2 12063.508} C_VEL
LIN {X 0,Y 514.601,Z 749.56,A -85,B 0,C 180,E1 12068.438,E2 12068.438} C_VEL
LIN {X 0,Y 514.342,Z 749.56,A -85,B 0,C 180,E1 12074.176,E2 12074.176} C_VEL
LIN {X 0,Y 514.18,Z 749.56,A -85,B 0,C 180,E1 12079.87,E2 12079.87} C_VEL
LIN {X 0,Y 513.994,Z 749.56,A -85,B 0,C 180,E1 12086.163,E2 12086.163} C_VEL
LIN {X 0,Y 513.854,Z 750.207,A -85,B 0,C 180,E1 12091.141,E2 12091.141} C_VEL
LIN {X 0,Y 516.436,Z 755.433,A -85,B 0,C 180,E1 12091.641,E2 12091.641} C_VEL
LIN {X 0,Y 540.514,Z 791.976,A -85,B 0,C 180,E1 12095.637,E2 12095.637} C_VEL
LIN {X 0,Y 566.523,Z 836.515,A -85,B 0,C 180,E1 12099.552,E2 12099.552} C_VEL
LIN {X 0,Y 574.212,Z 850.954,A -85,B 0,C 180,E1 12100.732,E2 12100.732} C_VEL
LIN {X 0,Y 568.603,Z 902.184,A -85,B 0,C 180,E1 12102.183,E2 12102.183} C_VEL
LIN {X 0,Y 562.078,Z 948.478,A -85,B 0,C 180,E1 12104.13,E2 12104.13} C_VEL
LIN {X 0,Y 554.011,Z 993.808,A -85,B 0,C 180,E1 12106.737,E2 12106.737} C_VEL
LIN {X 0,Y 545.597,Z 1036.026,A -85,B 0,C 180,E1 12109.893,E2 12109.893} C_VEL
LIN {X 0,Y 537.219,Z 1076.192,A -85,B 0,C 180,E1 12113.792,E2 12113.792} C_VEL
LIN {X 0,Y 530.151,Z 1110.195,A -85,B 0,C 180,E1 12117.934,E2 12117.934} C_VEL
LIN {X 0,Y 524.853,Z 1135.537,A -85,B 0,C 180,E1 12121.855,E2 12121.855} C_VEL
LIN {X 0,Y 523.641,Z 1142.016,A -85,B 0,C 180,E1 12123.043,E2 12123.043} C_VEL
LIN {X 0,Y 518.278,Z 1150.984,A -85,B 0,C 180,E1 12124.589,E2 12124.589} C_VEL
LIN {X 0,Y 512.867,Z 1159.335,A -85,B 0,C 180,E1 12126.199,E2 12126.199} C_VEL
LIN {X 0,Y 509.587,Z 1180.161,A -85,B 0,C 180,E1 12131.598,E2 12131.598} C_VEL
LIN {X 0,Y 507.777,Z 1195.37,A -85,B 0,C 180,E1 12137.102,E2 12137.102} C_VEL
LIN {X 0,Y 507.224,Z 1204.735,A -85,B 0,C 180,E1 12142.295,E2 12142.295} C_VEL
LIN {X 0,Y 507.067,Z 1208.889,A -85,B 0,C 180,E1 12146.582,E2 12146.582} C_VEL
LIN {X 0,Y 507.233,Z 1209.666,A -85,B 0,C 180,E1 12151.706,E2 12151.706} C_VEL
LIN {X 0,Y 507.174,Z 1205.911,A -85,B 0,C 180,E1 12156.844,E2 12156.844} C_VEL
LIN {X 0,Y 507.602,Z 1197.296,A -85,B 0,C 180,E1 12162.027,E2 12162.027} C_VEL
LIN {X 0,Y 509.005,Z 1183.702,A -85,B 0,C 180,E1 12167.269,E2 12167.269} C_VEL
LIN {X 0,Y 511.874,Z 1164.742,A -85,B 0,C 180,E1 12172.567,E2 12172.567} C_VEL
LIN {X 0,Y 516.855,Z 1139.218,A -85,B 0,C 180,E1 12177.89,E2 12177.89} C_VEL
LIN {X 0,Y 522.963,Z 1109.267,A -85,B 0,C 180,E1 12182.559,E2 12182.559} C_VEL
LIN {X 0,Y 530.935,Z 1071.987,A -85,B 0,C 180,E1 12187.08,E2 12187.08} C_VEL
LIN {X 0,Y 539.503,Z 1032.221,A -85,B 0,C 180,E1 12190.87,E2 12190.87} C_VEL
LIN {X 0,Y 549.15,Z 985.121,A -85,B 0,C 180,E1 12194.324,E2 12194.324} C_VEL
LIN {X 0,Y 557.225,Z 940.777,A -85,B 0,C 180,E1 12196.774,E2 12196.774} C_VEL
LIN {X 0,Y 564.218,Z 894.455,A -85,B 0,C 180,E1 12198.662,E2 12198.662} C_VEL
LIN {X 0,Y 568.501,Z 853.641,A -85,B 0,C 180,E1 12199.87,E2 12199.87} C_VEL
LIN {X 0,Y 548.592,Z 813.642,A -85,B 0,C 180,E1 12203.578,E2 12203.578} C_VEL
LIN {X 0,Y 531.207,Z 786.325,A -85,B 0,C 180,E1 12206.929,E2 12206.929} C_VEL
LIN {X 0,Y 514.563,Z 763.031,A -85,B 0,C 180,E1 12210.66,E2 12210.66} C_VEL
LIN {X 0,Y 509.36,Z 756.108,A -85,B 0,C 180,E1 12211.977,E2 12211.977} C_VEL
LIN {X 0,Y 506.067,Z 751.362,A -85,B 0,C 180,E1 12212.873,E2 12212.873} C_VEL
LIN {X 0,Y 505.877,Z 749.56,A -85,B 0,C 180,E1 12213.037,E2 12213.037} C_VEL
LIN {X 0,Y 506.039,Z 749.56,A -85,B 0,C 180,E1 12219.006,E2 12219.006} C_VEL
LIN {X 0,Y 506.339,Z 749.56,A -85,B 0,C 180,E1 12224.424,E2 12224.424} C_VEL
LIN {X 0,Y 506.616,Z 749.56,A -85,B 0,C 180,E1 12229.835,E2 12229.835} C_VEL
LIN {X 0,Y 506.888,Z 749.56,A -85,B 0,C 180,E1 12234.873,E2 12234.873} C_VEL
LIN {X 0,Y 507.139,Z 749.56,A -85,B 0,C 180,E1 12240.005,E2 12240.005} C_VEL
LIN {X 0,Y 506.815,Z 749.56,A -85,B 0,C 180,E1 12245.137,E2 12245.137} C_VEL
LIN {X 0,Y 506.582,Z 749.56,A -85,B 0,C 180,E1 12250.315,E2 12250.315} C_VEL
LIN {X 0,Y 506.154,Z 749.56,A -85,B 0,C 180,E1 12255.592,E2 12255.592} C_VEL
LIN {X 0,Y 505.956,Z 749.56,A -85,B 0,C 180,E1 12261.008,E2 12261.008} C_VEL
LIN {X 0,Y 505.942,Z 750.161,A -85,B 0,C 180,E1 12262.62,E2 12262.62} C_VEL
LIN {X 0,Y 508.325,Z 755.252,A -85,B 0,C 180,E1 12263.328,E2 12263.328} C_VEL
LIN {X 0,Y 511.303,Z 758.374,A -85,B 0,C 180,E1 12264.082,E2 12264.082} C_VEL
LIN {X 0,Y 529.942,Z 784.216,A -85,B 0,C 180,E1 12268.42,E2 12268.42} C_VEL
LIN {X 0,Y 547.999,Z 813.447,A -85,B 0,C 180,E1 12272.242,E2 12272.242} C_VEL
LIN {X 0,Y 561.797,Z 842.904,A -85,B 0,C 180,E1 12275.389,E2 12275.389} C_VEL
LIN {X 0,Y 563.165,Z 847.924,A -85,B 0,C 180,E1 12275.793,E2 12275.793} C_VEL
LIN {X 0,Y 556.25,Z 893.332,A -85,B 0,C 180,E1 12277.666,E2 12277.666} C_VEL
LIN {X 0,Y 548.211,Z 935.544,A -85,B 0,C 180,E1 12280.1,E2 12280.1} C_VEL
LIN {X 0,Y 539.049,Z 975.776,A -85,B 0,C 180,E1 12283.21,E2 12283.21} C_VEL
LIN {X 0,Y 530.587,Z 1010.433,A -85,B 0,C 180,E1 12286.721,E2 12286.721} C_VEL
LIN {X 0,Y 522.307,Z 1043.773,A -85,B 0,C 180,E1 12291.083,E2 12291.083} C_VEL
LIN {X 0,Y 515.404,Z 1073.041,A -85,B 0,C 180,E1 12296.148,E2 12296.148} C_VEL
LIN {X 0,Y 511.07,Z 1094.751,A -85,B 0,C 180,E1 12301.139,E2 12301.139} C_VEL
LIN {X 0,Y 508.645,Z 1111.522,A -85,B 0,C 180,E1 12306.357,E2 12306.357} C_VEL
LIN {X 0,Y 507.384,Z 1122.992,A -85,B 0,C 180,E1 12311.723,E2 12311.723} C_VEL
LIN {X 0,Y 506.87,Z 1128.62,A -85,B 0,C 180,E1 12316.203,E2 12316.203} C_VEL
LIN {X 0,Y 506.834,Z 1130.604,A -85,B 0,C 180,E1 12321.428,E2 12321.428} C_VEL
LIN {X 0,Y 507.182,Z 1127.749,A -85,B 0,C 180,E1 12326.585,E2 12326.585} C_VEL
LIN {X 0,Y 507.66,Z 1120.257,A -85,B 0,C 180,E1 12331.707,E2 12331.707} C_VEL
LIN {X 0,Y 509.081,Z 1107.753,A -85,B 0,C 180,E1 12336.82,E2 12336.82} C_VEL
LIN {X 0,Y 511.872,Z 1090.046,A -85,B 0,C 180,E1 12341.927,E2 12341.927} C_VEL
LIN {X 0,Y 517.027,Z 1065.062,A -85,B 0,C 180,E1 12347.214,E2 12347.214} C_VEL
LIN {X 0,Y 523.754,Z 1036.081,A -85,B 0,C 180,E1 12351.807,E2 12351.807} C_VEL
LIN {X 0,Y 531.498,Z 1003.383,A -85,B 0,C 180,E1 12355.815,E2 12355.815} C_VEL
LIN {X 0,Y 540.311,Z 964.867,A -85,B 0,C 180,E1 12359.419,E2 12359.419} C_VEL
LIN {X 0,Y 548.469,Z 924.771,A -85,B 0,C 180,E1 12362.244,E2 12362.244} C_VEL
LIN {X 0,Y 555.72,Z 882.626,A -85,B 0,C 180,E1 12364.468,E2 12364.468} C_VEL
LIN {X 0,Y 560.218,Z 844.836,A -85,B 0,C 180,E1 12365.971,E2 12365.971} C_VEL
LIN {X 0,Y 540.87,Z 806.289,A -85,B 0,C 180,E1 12369.631,E2 12369.631} C_VEL
LIN {X 0,Y 517.939,Z 768.853,A -85,B 0,C 180,E1 12373.612,E2 12373.612} C_VEL
LIN {X 0,Y 507.985,Z 755.113,A -85,B 0,C 180,E1 12375.401,E2 12375.401} C_VEL
LIN {X 0,Y 505.646,Z 749.56,A -85,B 0,C 180,E1 12376.023,E2 12376.023} C_VEL
LIN {X 0,Y 505.681,Z 749.56,A -85,B 0,C 180,E1 12381.124,E2 12381.124} C_VEL
LIN {X 0,Y 505.669,Z 749.56,A -85,B 0,C 180,E1 12387.452,E2 12387.452} C_VEL
LIN {X 0,Y 505.872,Z 749.56,A -85,B 0,C 180,E1 12393.659,E2 12393.659} C_VEL
LIN {X 0,Y 505.946,Z 749.56,A -85,B 0,C 180,E1 12398.992,E2 12398.992} C_VEL
LIN {X 0,Y 506.152,Z 749.56,A -85,B 0,C 180,E1 12404.408,E2 12404.408} C_VEL
LIN {X 0,Y 506.628,Z 749.56,A -85,B 0,C 180,E1 12409.837,E2 12409.837} C_VEL
LIN {X 0,Y 506.826,Z 749.56,A -85,B 0,C 180,E1 12414.863,E2 12414.863} C_VEL
LIN {X 0,Y 507.149,Z 749.56,A -85,B 0,C 180,E1 12419.995,E2 12419.995} C_VEL
LIN {X 0,Y 506.899,Z 749.56,A -85,B 0,C 180,E1 12425.126,E2 12425.126} C_VEL
LIN {X 0,Y 506.594,Z 749.56,A -85,B 0,C 180,E1 12430.306,E2 12430.306} C_VEL
LIN {X 0,Y 506.412,Z 749.56,A -85,B 0,C 180,E1 12435.574,E2 12435.574} C_VEL
LIN {X 0,Y 506.202,Z 749.56,A -85,B 0,C 180,E1 12440.987,E2 12440.987} C_VEL
LIN {X 0,Y 506.039,Z 749.56,A -85,B 0,C 180,E1 12446.606,E2 12446.606} C_VEL
LIN {X 0,Y 505.939,Z 749.648,A -85,B 0,C 180,E1 12449.915,E2 12449.915} C_VEL
LIN {X 0,Y 508.219,Z 755.146,A -85,B 0,C 180,E1 12450.403,E2 12450.403} C_VEL
LIN {X 0,Y 511.049,Z 759.162,A -85,B 0,C 180,E1 12450.929,E2 12450.929} C_VEL
LIN {X 0,Y 533.315,Z 792.639,A -85,B 0,C 180,E1 12454.748,E2 12454.748} C_VEL
LIN {X 0,Y 560.269,Z 838.777,A -85,B 0,C 180,E1 12458.955,E2 12458.955} C_VEL
LIN {X 0,Y 568.346,Z 855.137,A -85,B 0,C 180,E1 12460.282,E2 12460.282} C_VEL
LIN {X 0,Y 562.504,Z 904.823,A -85,B 0,C 180,E1 12461.722,E2 12461.722} C_VEL
LIN {X 0,Y 555.915,Z 949.235,A -85,B 0,C 180,E1 12463.627,E2 12463.627} C_VEL
LIN {X 0,Y 547.578,Z 994.613,A -85,B 0,C 180,E1 12466.266,E2 12466.266} C_VEL
LIN {X 0,Y 538.892,Z 1036.429,A -85,B 0,C 180,E1 12469.44,E2 12469.44} C_VEL
LIN {X 0,Y 529.81,Z 1078.111,A -85,B 0,C 180,E1 12473.559,E2 12473.559} C_VEL
LIN {X 0,Y 522.358,Z 1112.46,A -85,B 0,C 180,E1 12477.887,E2 12477.887} C_VEL
LIN {X 0,Y 516.24,Z 1142.139,A -85,B 0,C 180,E1 12482.649,E2 12482.649} C_VEL
LIN {X 0,Y 512.867,Z 1159.335,A -85,B 0,C 180,E1 12486.199,E2 12486.199} C_VEL
LIN {X 0,Y 507.637,Z 1167.168,A -85,B 0,C 180,E1 12487.863,E2 12487.863} C_VEL
LIN {X 0,Y 502.641,Z 1174.326,A -85,B 0,C 180,E1 12489.593,E2 12489.593} C_VEL
LIN {X 0,Y 500.435,Z 1190.977,A -85,B 0,C 180,E1 12495.065,E2 12495.065} C_VEL
LIN {X 0,Y 499.431,Z 1202.212,A -85,B 0,C 180,E1 12500.42,E2 12500.42} C_VEL
LIN {X 0,Y 499.162,Z 1207.641,A -85,B 0,C 180,E1 12504.788,E2 12504.788} C_VEL
LIN {X 0,Y 499.235,Z 1210,A -85,B 0,C 180,E1 12509.999,E2 12509.999} C_VEL
LIN {X 0,Y 499.156,Z 1207.644,A -85,B 0,C 180,E1 12515.21,E2 12515.21} C_VEL
LIN {X 0,Y 499.522,Z 1200.655,A -85,B 0,C 180,E1 12520.457,E2 12520.457} C_VEL
LIN {X 0,Y 500.642,Z 1188.849,A -85,B 0,C 180,E1 12525.762,E2 12525.762} C_VEL
LIN {X 0,Y 503.077,Z 1171.688,A -85,B 0,C 180,E1 12531.127,E2 12531.127} C_VEL
LIN {X 0,Y 507.125,Z 1149.449,A -85,B 0,C 180,E1 12536.31,E2 12536.31} C_VEL
LIN {X 0,Y 513.18,Z 1120.584,A -85,B 0,C 180,E1 12541.283,E2 12541.283} C_VEL
LIN {X 0,Y 521.109,Z 1084.988,A -85,B 0,C 180,E1 12546.048,E2 12546.048} C_VEL
LIN {X 0,Y 529.737,Z 1046.831,A -85,B 0,C 180,E1 12550.062,E2 12550.062} C_VEL
LIN {X 0,Y 539.469,Z 1002.934,A -85,B 0,C 180,E1 12553.655,E2 12553.655} C_VEL
LIN {X 0,Y 547.948,Z 960.22,A -85,B 0,C 180,E1 12556.356,E2 12556.356} C_VEL
LIN {X 0,Y 556.013,Z 912.889,A -85,B 0,C 180,E1 12558.592,E2 12558.592} C_VEL
LIN {X 0,Y 562.455,Z 865.286,A -85,B 0,C 180,E1 12560.14,E2 12560.14} C_VEL
LIN {X 0,Y 562.692,Z 856.599,A -85,B 0,C 180,E1 12560.438,E2 12560.438} C_VEL
LIN {X 0,Y 544.768,Z 819.449,A -85,B 0,C 180,E1 12563.975,E2 12563.975} C_VEL
LIN {X 0,Y 528.152,Z 792.826,A -85,B 0,C 180,E1 12567.288,E2 12567.288} C_VEL
LIN {X 0,Y 511.815,Z 769.831,A -85,B 0,C 180,E1 12571.032,E2 12571.032} C_VEL
LIN {X 0,Y 506.34,Z 762.667,A -85,B 0,C 180,E1 12572.451,E2 12572.451} C_VEL
LIN {X 0,Y 501.949,Z 756.386,A -85,B 0,C 180,E1 12573.687,E2 12573.687} C_VEL
LIN {X 0,Y 498.247,Z 751.67,A -85,B 0,C 180,E1 12574.779,E2 12574.779} C_VEL
LIN {X 0,Y 497.982,Z 749.56,A -85,B 0,C 180,E1 12575.058,E2 12575.058} C_VEL
LIN {X 0,Y 498.209,Z 749.56,A -85,B 0,C 180,E1 12580.515,E2 12580.515} C_VEL
LIN {X 0,Y 498.527,Z 749.56,A -85,B 0,C 180,E1 12585.971,E2 12585.971} C_VEL
LIN {X 0,Y 498.751,Z 749.56,A -85,B 0,C 180,E1 12591.291,E2 12591.291} C_VEL
LIN {X 0,Y 498.99,Z 749.56,A -85,B 0,C 180,E1 12596.532,E2 12596.532} C_VEL
LIN {X 0,Y 499.07,Z 749.56,A -85,B 0,C 180,E1 12601.74,E2 12601.74} C_VEL
LIN {X 0,Y 498.82,Z 749.56,A -85,B 0,C 180,E1 12606.965,E2 12606.965} C_VEL
LIN {X 0,Y 498.507,Z 749.56,A -85,B 0,C 180,E1 12612.256,E2 12612.256} C_VEL
LIN {X 0,Y 498.127,Z 749.56,A -85,B 0,C 180,E1 12617.665,E2 12617.665} C_VEL
LIN {X 0,Y 498.058,Z 749.925,A -85,B 0,C 180,E1 12620.658,E2 12620.658} C_VEL
LIN {X 0,Y 500.121,Z 754.921,A -85,B 0,C 180,E1 12621.36,E2 12621.36} C_VEL
LIN {X 0,Y 503.518,Z 758.238,A -85,B 0,C 180,E1 12622.304,E2 12622.304} C_VEL
LIN {X 0,Y 507.957,Z 763.878,A -85,B 0,C 180,E1 12623.51,E2 12623.51} C_VEL
LIN {X 0,Y 527.265,Z 791.535,A -85,B 0,C 180,E1 12628.169,E2 12628.169} C_VEL
LIN {X 0,Y 544.273,Z 819.901,A -85,B 0,C 180,E1 12631.961,E2 12631.961} C_VEL
LIN {X 0,Y 557.33,Z 848.981,A -85,B 0,C 180,E1 12635.106,E2 12635.106} C_VEL
LIN {X 0,Y 557.227,Z 854.44,A -85,B 0,C 180,E1 12635.389,E2 12635.389} C_VEL
LIN {X 0,Y 549.725,Z 900.709,A -85,B 0,C 180,E1 12637.397,E2 12637.397} C_VEL
LIN {X 0,Y 540.953,Z 943.044,A -85,B 0,C 180,E1 12639.985,E2 12639.985} C_VEL
LIN {X 0,Y 531.854,Z 981.192,A -85,B 0,C 180,E1 12643.071,E2 12643.071} C_VEL
LIN {X 0,Y 522.282,Z 1018.198,A -85,B 0,C 180,E1 12647.026,E2 12647.026} C_VEL
LIN {X 0,Y 514.397,Z 1048.354,A -85,B 0,C 180,E1 12651.222,E2 12651.222} C_VEL
LIN {X 0,Y 507.719,Z 1075.694,A -85,B 0,C 180,E1 12656.136,E2 12656.136} C_VEL
LIN {X 0,Y 502.956,Z 1098.915,A -85,B 0,C 180,E1 12661.764,E2 12661.764} C_VEL
LIN {X 0,Y 500.631,Z 1114.097,A -85,B 0,C 180,E1 12666.897,E2 12666.897} C_VEL
LIN {X 0,Y 499.433,Z 1125.028,A -85,B 0,C 180,E1 12672.389,E2 12672.389} C_VEL
LIN {X 0,Y 498.88,Z 1130.381,A -85,B 0,C 180,E1 12677.759,E2 12677.759} C_VEL
LIN {X 0,Y 499.067,Z 1130.947,A -85,B 0,C 180,E1 12683.044,E2 12683.044} C_VEL
LIN {X 0,Y 499.35,Z 1126.594,A -85,B 0,C 180,E1 12688.267,E2 12688.267} C_VEL
LIN {X 0,Y 499.983,Z 1119.423,A -85,B 0,C 180,E1 12692.599,E2 12692.599} C_VEL
LIN {X 0,Y 501.716,Z 1106.375,A -85,B 0,C 180,E1 12697.791,E2 12697.791} C_VEL
LIN {X 0,Y 505.121,Z 1086.899,A -85,B 0,C 180,E1 12703.181,E2 12703.181} C_VEL
LIN {X 0,Y 510.476,Z 1062.967,A -85,B 0,C 180,E1 12708.11,E2 12708.11} C_VEL
LIN {X 0,Y 517.827,Z 1033.069,A -85,B 0,C 180,E1 12712.783,E2 12712.783} C_VEL
LIN {X 0,Y 526.168,Z 998.972,A -85,B 0,C 180,E1 12716.842,E2 12716.842} C_VEL
LIN {X 0,Y 534.87,Z 961.535,A -85,B 0,C 180,E1 12720.268,E2 12720.268} C_VEL
LIN {X 0,Y 543.873,Z 918.272,A -85,B 0,C 180,E1 12723.23,E2 12723.23} C_VEL
LIN {X 0,Y 550.814,Z 877.479,A -85,B 0,C 180,E1 12725.276,E2 12725.276} C_VEL
LIN {X 0,Y 554.329,Z 848.096,A -85,B 0,C 180,E1 12726.461,E2 12726.461} C_VEL
LIN {X 0,Y 534.477,Z 808.255,A -85,B 0,C 180,E1 12730.358,E2 12730.358} C_VEL
LIN {X 0,Y 513.161,Z 773.713,A -85,B 0,C 180,E1 12734.196,E2 12734.196} C_VEL
LIN {X 0,Y 500.287,Z 755.346,A -85,B 0,C 180,E1 12736.618,E2 12736.618} C_VEL
LIN {X 0,Y 497.807,Z 750.678,A -85,B 0,C 180,E1 12737.143,E2 12737.143} C_VEL
LIN {X 0,Y 497.705,Z 749.56,A -85,B 0,C 180,E1 12737.349,E2 12737.349} C_VEL
LIN {X 0,Y 497.721,Z 749.56,A -85,B 0,C 180,E1 12742.604,E2 12742.604} C_VEL
LIN {X 0,Y 497.759,Z 749.56,A -85,B 0,C 180,E1 12748.923,E2 12748.923} C_VEL
LIN {X 0,Y 497.928,Z 749.56,A -85,B 0,C 180,E1 12754.851,E2 12754.851} C_VEL
LIN {X 0,Y 498.077,Z 749.56,A -85,B 0,C 180,E1 12760.499,E2 12760.499} C_VEL
LIN {X 0,Y 498.371,Z 749.56,A -85,B 0,C 180,E1 12766,E2 12766} C_VEL
LIN {X 0,Y 498.764,Z 749.56,A -85,B 0,C 180,E1 12771.282,E2 12771.282} C_VEL
LIN {X 0,Y 499.096,Z 749.56,A -85,B 0,C 180,E1 12776.523,E2 12776.523} C_VEL
LIN {X 0,Y 499.065,Z 749.56,A -85,B 0,C 180,E1 12782.251,E2 12782.251} C_VEL
LIN {X 0,Y 498.864,Z 749.56,A -85,B 0,C 180,E1 12786.955,E2 12786.955} C_VEL
LIN {X 0,Y 498.58,Z 749.56,A -85,B 0,C 180,E1 12792.244,E2 12792.244} C_VEL
LIN {X 0,Y 498.415,Z 749.56,A -85,B 0,C 180,E1 12797.644,E2 12797.644} C_VEL
LIN {X 0,Y 498.171,Z 749.56,A -85,B 0,C 180,E1 12803.22,E2 12803.22} C_VEL
LIN {X 0,Y 498.115,Z 750.354,A -85,B 0,C 180,E1 12808.664,E2 12808.664} C_VEL
LIN {X 0,Y 500.689,Z 755.484,A -85,B 0,C 180,E1 12809.216,E2 12809.216} C_VEL
LIN {X 0,Y 519.006,Z 782.306,A -85,B 0,C 180,E1 12812.612,E2 12812.612} C_VEL
LIN {X 0,Y 544.568,Z 824.001,A -85,B 0,C 180,E1 12816.809,E2 12816.809} C_VEL
LIN {X 0,Y 562.441,Z 857.802,A -85,B 0,C 180,E1 12819.771,E2 12819.771} C_VEL
LIN {X 0,Y 556.595,Z 905.953,A -85,B 0,C 180,E1 12821.198,E2 12821.198} C_VEL
LIN {X 0,Y 549.724,Z 950.346,A -85,B 0,C 180,E1 12823.136,E2 12823.136} C_VEL
LIN {X 0,Y 541.041,Z 995.933,A -85,B 0,C 180,E1 12825.822,E2 12825.822} C_VEL
LIN {X 0,Y 531.988,Z 1037.702,A -85,B 0,C 180,E1 12829.051,E2 12829.051} C_VEL
LIN {X 0,Y 522.545,Z 1079.442,A -85,B 0,C 180,E1 12833.255,E2 12833.255} C_VEL
LIN {X 0,Y 514.852,Z 1113.315,A -85,B 0,C 180,E1 12837.632,E2 12837.632} C_VEL
LIN {X 0,Y 508.341,Z 1144.503,A -85,B 0,C 180,E1 12842.733,E2 12842.733} C_VEL
LIN {X 0,Y 504.019,Z 1166.299,A -85,B 0,C 180,E1 12847.475,E2 12847.475} C_VEL
LIN {X 0,Y 502.641,Z 1174.326,A -85,B 0,C 180,E1 12849.593,E2 12849.593} C_VEL
LIN {X 0,Y 497.782,Z 1180.919,A -85,B 0,C 180,E1 12851.378,E2 12851.378} C_VEL
LIN {X 0,Y 493.088,Z 1186.76,A -85,B 0,C 180,E1 12853.212,E2 12853.212} C_VEL
LIN {X 0,Y 491.816,Z 1199.087,A -85,B 0,C 180,E1 12858.479,E2 12858.479} C_VEL
LIN {X 0,Y 491.403,Z 1205.908,A -85,B 0,C 180,E1 12862.934,E2 12862.934} C_VEL
LIN {X 0,Y 491.219,Z 1209.665,A -85,B 0,C 180,E1 12868.236,E2 12868.236} C_VEL
LIN {X 0,Y 491.434,Z 1209.666,A -85,B 0,C 180,E1 12871.761,E2 12871.761} C_VEL
LIN {X 0,Y 491.388,Z 1205.911,A -85,B 0,C 180,E1 12877.065,E2 12877.065} C_VEL
LIN {X 0,Y 491.885,Z 1197.29,A -85,B 0,C 180,E1 12882.417,E2 12882.417} C_VEL
LIN {X 0,Y 493.499,Z 1183.701,A -85,B 0,C 180,E1 12887.83,E2 12887.83} C_VEL
LIN {X 0,Y 496.762,Z 1164.732,A -85,B 0,C 180,E1 12893.293,E2 12893.293} C_VEL
LIN {X 0,Y 501.801,Z 1138.938,A -85,B 0,C 180,E1 12898.558,E2 12898.558} C_VEL
LIN {X 0,Y 508.599,Z 1108.257,A -85,B 0,C 180,E1 12903.47,E2 12903.47} C_VEL
LIN {X 0,Y 517.062,Z 1071.943,A -85,B 0,C 180,E1 12907.991,E2 12907.991} C_VEL
LIN {X 0,Y 526.426,Z 1032.467,A -85,B 0,C 180,E1 12911.878,E2 12911.878} C_VEL
LIN {X 0,Y 536.921,Z 985.533,A -85,B 0,C 180,E1 12915.424,E2 12915.424} C_VEL
LIN {X 0,Y 545.621,Z 942.341,A -85,B 0,C 180,E1 12917.877,E2 12917.877} C_VEL
LIN {X 0,Y 553.001,Z 897.566,A -85,B 0,C 180,E1 12919.762,E2 12919.762} C_VEL
LIN {X 0,Y 557.388,Z 860.474,A -85,B 0,C 180,E1 12920.93,E2 12920.93} C_VEL
LIN {X 0,Y 540.289,Z 823.96,A -85,B 0,C 180,E1 12924.514,E2 12924.514} C_VEL
LIN {X 0,Y 523.047,Z 796.071,A -85,B 0,C 180,E1 12928.107,E2 12928.107} C_VEL
LIN {X 0,Y 507.946,Z 775.19,A -85,B 0,C 180,E1 12931.701,E2 12931.701} C_VEL
LIN {X 0,Y 502.8,Z 768.351,A -85,B 0,C 180,E1 12933.088,E2 12933.088} C_VEL
LIN {X 0,Y 499.156,Z 763.196,A -85,B 0,C 180,E1 12934.147,E2 12934.147} C_VEL
LIN {X 0,Y 495.4,Z 757.262,A -85,B 0,C 180,E1 12935.328,E2 12935.328} C_VEL
LIN {X 0,Y 490.659,Z 752.483,A -85,B 0,C 180,E1 12936.835,E2 12936.835} C_VEL
LIN {X 0,Y 490.098,Z 749.56,A -85,B 0,C 180,E1 12937.238,E2 12937.238} C_VEL
LIN {X 0,Y 490.386,Z 749.56,A -85,B 0,C 180,E1 12942.795,E2 12942.795} C_VEL
LIN {X 0,Y 490.641,Z 749.56,A -85,B 0,C 180,E1 12947.554,E2 12947.554} C_VEL
LIN {X 0,Y 490.941,Z 749.56,A -85,B 0,C 180,E1 12952.932,E2 12952.932} C_VEL
LIN {X 0,Y 491.259,Z 749.56,A -85,B 0,C 180,E1 12958.242,E2 12958.242} C_VEL
LIN {X 0,Y 491.166,Z 749.56,A -85,B 0,C 180,E1 12963.533,E2 12963.533} C_VEL
LIN {X 0,Y 490.735,Z 749.56,A -85,B 0,C 180,E1 12969.815,E2 12969.815} C_VEL
LIN {X 0,Y 490.276,Z 749.56,A -85,B 0,C 180,E1 12976.11,E2 12976.11} C_VEL
LIN {X 0,Y 490.164,Z 749.56,A -85,B 0,C 180,E1 12978.427,E2 12978.427} C_VEL
LIN {X 0,Y 491.835,Z 754.435,A -85,B 0,C 180,E1 12979.117,E2 12979.117} C_VEL
LIN {X 0,Y 495.876,Z 758.318,A -85,B 0,C 180,E1 12980.377,E2 12980.377} C_VEL
LIN {X 0,Y 500.152,Z 763.912,A -85,B 0,C 180,E1 12981.67,E2 12981.67} C_VEL
LIN {X 0,Y 516.802,Z 787.224,A -85,B 0,C 180,E1 12986.079,E2 12986.079} C_VEL
LIN {X 0,Y 533.524,Z 813.286,A -85,B 0,C 180,E1 12990.012,E2 12990.012} C_VEL
LIN {X 0,Y 548.338,Z 843.368,A -85,B 0,C 180,E1 12993.631,E2 12993.631} C_VEL
LIN {X 0,Y 552.208,Z 854.741,A -85,B 0,C 180,E1 12994.751,E2 12994.751} C_VEL
LIN {X 0,Y 544.399,Z 901.4,A -85,B 0,C 180,E1 12996.784,E2 12996.784} C_VEL
LIN {X 0,Y 535.247,Z 943.954,A -85,B 0,C 180,E1 12999.404,E2 12999.404} C_VEL
LIN {X 0,Y 525.819,Z 981.933,A -85,B 0,C 180,E1 13002.503,E2 13002.503} C_VEL
LIN {X 0,Y 515.794,Z 1018.926,A -85,B 0,C 180,E1 13006.492,E2 13006.492} C_VEL
LIN {X 0,Y 507.239,Z 1050.079,A -85,B 0,C 180,E1 13010.901,E2 13010.901} C_VEL
LIN {X 0,Y 500.411,Z 1076.545,A -85,B 0,C 180,E1 13015.755,E2 13015.755} C_VEL
LIN {X 0,Y 495.52,Z 1098.805,A -85,B 0,C 180,E1 13021.222,E2 13021.222} C_VEL
LIN {X 0,Y 492.949,Z 1114.425,A -85,B 0,C 180,E1 13026.516,E2 13026.516} C_VEL
LIN {X 0,Y 491.61,Z 1125.456,A -85,B 0,C 180,E1 13032.099,E2 13032.099} C_VEL
LIN {X 0,Y 491.006,Z 1130.958,A -85,B 0,C 180,E1 13037.56,E2 13037.56} C_VEL
LIN {X 0,Y 491.171,Z 1131.622,A -85,B 0,C 180,E1 13042.932,E2 13042.932} C_VEL
LIN {X 0,Y 491.512,Z 1127.426,A -85,B 0,C 180,E1 13048.239,E2 13048.239} C_VEL
LIN {X 0,Y 492.17,Z 1120.374,A -85,B 0,C 180,E1 13052.641,E2 13052.641} C_VEL
LIN {X 0,Y 493.972,Z 1107.458,A -85,B 0,C 180,E1 13057.913,E2 13057.913} C_VEL
LIN {X 0,Y 497.504,Z 1088.3,A -85,B 0,C 180,E1 13063.36,E2 13063.36} C_VEL
LIN {X 0,Y 502.983,Z 1065.001,A -85,B 0,C 180,E1 13068.288,E2 13068.288} C_VEL
LIN {X 0,Y 510.941,Z 1033.836,A -85,B 0,C 180,E1 13073.239,E2 13073.239} C_VEL
LIN {X 0,Y 519.609,Z 999.694,A -85,B 0,C 180,E1 13077.347,E2 13077.347} C_VEL
LIN {X 0,Y 528.518,Z 962.817,A -85,B 0,C 180,E1 13080.759,E2 13080.759} C_VEL
LIN {X 0,Y 537.698,Z 920.183,A -85,B 0,C 180,E1 13083.714,E2 13083.714} C_VEL
LIN {X 0,Y 545.057,Z 878.675,A -85,B 0,C 180,E1 13085.824,E2 13085.824} C_VEL
LIN {X 0,Y 548.405,Z 851.451,A -85,B 0,C 180,E1 13086.947,E2 13086.947} C_VEL
LIN {X 0,Y 529.124,Z 812.239,A -85,B 0,C 180,E1 13090.909,E2 13090.909} C_VEL
LIN {X 0,Y 509.719,Z 780.046,A -85,B 0,C 180,E1 13094.558,E2 13094.558} C_VEL
LIN {X 0,Y 492.613,Z 755.539,A -85,B 0,C 180,E1 13097.907,E2 13097.907} C_VEL
LIN {X 0,Y 489.93,Z 750.768,A -85,B 0,C 180,E1 13098.501,E2 13098.501} C_VEL
LIN {X 0,Y 489.832,Z 749.56,A -85,B 0,C 180,E1 13098.585,E2 13098.585} C_VEL
LIN {X 0,Y 489.773,Z 749.56,A -85,B 0,C 180,E1 13104.104,E2 13104.104} C_VEL
LIN {X 0,Y 489.857,Z 749.56,A -85,B 0,C 180,E1 13110.418,E2 13110.418} C_VEL
LIN {X 0,Y 490.024,Z 749.56,A -85,B 0,C 180,E1 13116.36,E2 13116.36} C_VEL
LIN {X 0,Y 490.204,Z 749.56,A -85,B 0,C 180,E1 13122.87,E2 13122.87} C_VEL
LIN {X 0,Y 490.745,Z 749.56,A -85,B 0,C 180,E1 13129.348,E2 13129.348} C_VEL
LIN {X 0,Y 491.004,Z 749.56,A -85,B 0,C 180,E1 13134.697,E2 13134.697} C_VEL
LIN {X 0,Y 491.355,Z 749.56,A -85,B 0,C 180,E1 13139.995,E2 13139.995} C_VEL
LIN {X 0,Y 491.087,Z 749.56,A -85,B 0,C 180,E1 13145.292,E2 13145.292} C_VEL
LIN {X 0,Y 490.756,Z 749.56,A -85,B 0,C 180,E1 13150.642,E2 13150.642} C_VEL
LIN {X 0,Y 490.538,Z 749.56,A -85,B 0,C 180,E1 13156.091,E2 13156.091} C_VEL
LIN {X 0,Y 490.252,Z 749.56,A -85,B 0,C 180,E1 13162.374,E2 13162.374} C_VEL
LIN {X 0,Y 490.185,Z 749.956,A -85,B 0,C 180,E1 13167.285,E2 13167.285} C_VEL
LIN {X 0,Y 492.587,Z 755.282,A -85,B 0,C 180,E1 13167.846,E2 13167.846} C_VEL
LIN {X 0,Y 495.202,Z 758.747,A -85,B 0,C 180,E1 13168.385,E2 13168.385} C_VEL
LIN {X 0,Y 516.323,Z 789.995,A -85,B 0,C 180,E1 13172.404,E2 13172.404} C_VEL
LIN {X 0,Y 540.884,Z 830.695,A -85,B 0,C 180,E1 13176.539,E2 13176.539} C_VEL
LIN {X 0,Y 556.483,Z 861.07,A -85,B 0,C 180,E1 13179.261,E2 13179.261} C_VEL
LIN {X 0,Y 550.34,Z 909.879,A -85,B 0,C 180,E1 13180.772,E2 13180.772} C_VEL
LIN {X 0,Y 542.841,Z 955.224,A -85,B 0,C 180,E1 13182.832,E2 13182.832} C_VEL
LIN {X 0,Y 533.957,Z 1000.062,A -85,B 0,C 180,E1 13185.56,E2 13185.56} C_VEL
LIN {X 0,Y 524.175,Z 1042.896,A -85,B 0,C 180,E1 13189.015,E2 13189.015} C_VEL
LIN {X 0,Y 515.104,Z 1081.448,A -85,B 0,C 180,E1 13193.029,E2 13193.029} C_VEL
LIN {X 0,Y 506.506,Z 1117.679,A -85,B 0,C 180,E1 13197.889,E2 13197.889} C_VEL
LIN {X 0,Y 500.331,Z 1146.395,A -85,B 0,C 180,E1 13202.81,E2 13202.81} C_VEL
LIN {X 0,Y 496.036,Z 1168.217,A -85,B 0,C 180,E1 13207.616,E2 13207.616} C_VEL
LIN {X 0,Y 493.14,Z 1186.361,A -85,B 0,C 180,E1 13213.075,E2 13213.075} C_VEL
LIN {X 0,Y 493.088,Z 1186.76,A -85,B 0,C 180,E1 13213.212,E2 13213.212} C_VEL
LIN {X 0,Y 488.544,Z 1192.002,A -85,B 0,C 180,E1 13215.091,E2 13215.091} C_VEL
LIN {X 0,Y 484.116,Z 1196.55,A -85,B 0,C 180,E1 13217.028,E2 13217.028} C_VEL
LIN {X 0,Y 483.542,Z 1204.726,A -85,B 0,C 180,E1 13221.915,E2 13221.915} C_VEL
LIN {X 0,Y 483.372,Z 1208.881,A -85,B 0,C 180,E1 13226.414,E2 13226.414} C_VEL
LIN {X 0,Y 483.549,Z 1209.666,A -85,B 0,C 180,E1 13231.79,E2 13231.79} C_VEL
LIN {X 0,Y 483.487,Z 1205.911,A -85,B 0,C 180,E1 13237.181,E2 13237.181} C_VEL
LIN {X 0,Y 484.025,Z 1197.287,A -85,B 0,C 180,E1 13242.622,E2 13242.622} C_VEL
LIN {X 0,Y 485.769,Z 1183.7,A -85,B 0,C 180,E1 13248.123,E2 13248.123} C_VEL
LIN {X 0,Y 488.395,Z 1167.725,A -85,B 0,C 180,E1 13252.752,E2 13252.752} C_VEL
LIN {X 0,Y 493.379,Z 1143.193,A -85,B 0,C 180,E1 13258.092,E2 13258.092} C_VEL
LIN {X 0,Y 500.368,Z 1112.171,A -85,B 0,C 180,E1 13263.283,E2 13263.283} C_VEL
LIN {X 0,Y 508.571,Z 1078.823,A -85,B 0,C 180,E1 13267.689,E2 13267.689} C_VEL
LIN {X 0,Y 518.984,Z 1036.63,A -85,B 0,C 180,E1 13272.042,E2 13272.042} C_VEL
LIN {X 0,Y 529.118,Z 994.243,A -85,B 0,C 180,E1 13275.413,E2 13275.413} C_VEL
LIN {X 0,Y 538.425,Z 950.749,A -85,B 0,C 180,E1 13278.057,E2 13278.057} C_VEL
LIN {X 0,Y 546.394,Z 906.848,A -85,B 0,C 180,E1 13280.048,E2 13280.048} C_VEL
LIN {X 0,Y 551.909,Z 864.029,A -85,B 0,C 180,E1 13281.477,E2 13281.477} C_VEL
LIN {X 0,Y 536.365,Z 829.547,A -85,B 0,C 180,E1 13284.939,E2 13284.939} C_VEL
LIN {X 0,Y 519.865,Z 802.322,A -85,B 0,C 180,E1 13288.525,E2 13288.525} C_VEL
LIN {X 0,Y 502.406,Z 777.492,A -85,B 0,C 180,E1 13292.884,E2 13292.884} C_VEL
LIN {X 0,Y 495.935,Z 769.389,A -85,B 0,C 180,E1 13294.754,E2 13294.754} C_VEL
LIN {X 0,Y 491.913,Z 763.687,A -85,B 0,C 180,E1 13296.046,E2 13296.046} C_VEL
LIN {X 0,Y 487.984,Z 758.151,A -85,B 0,C 180,E1 13297.406,E2 13297.406} C_VEL
LIN {X 0,Y 482.66,Z 752.064,A -85,B 0,C 180,E1 13299.382,E2 13299.382} C_VEL
LIN {X 0,Y 482.319,Z 749.56,A -85,B 0,C 180,E1 13299.726,E2 13299.726} C_VEL
LIN {X 0,Y 482.68,Z 749.56,A -85,B 0,C 180,E1 13306.049,E2 13306.049} C_VEL
LIN {X 0,Y 482.933,Z 749.56,A -85,B 0,C 180,E1 13311.004,E2 13311.004} C_VEL
LIN {X 0,Y 483.184,Z 749.56,A -85,B 0,C 180,E1 13316.419,E2 13316.419} C_VEL
LIN {X 0,Y 483.297,Z 749.56,A -85,B 0,C 180,E1 13321.797,E2 13321.797} C_VEL
LIN {X 0,Y 482.988,Z 749.56,A -85,B 0,C 180,E1 13327.194,E2 13327.194} C_VEL
LIN {X 0,Y 482.635,Z 749.56,A -85,B 0,C 180,E1 13332.666,E2 13332.666} C_VEL
LIN {X 0,Y 482.417,Z 750.158,A -85,B 0,C 180,E1 13335.971,E2 13335.971} C_VEL
LIN {X 0,Y 484.5,Z 755.011,A -85,B 0,C 180,E1 13336.89,E2 13336.89} C_VEL
LIN {X 0,Y 488.087,Z 758.256,A -85,B 0,C 180,E1 13338.157,E2 13338.157} C_VEL
LIN {X 0,Y 492.022,Z 763.696,A -85,B 0,C 180,E1 13339.517,E2 13339.517} C_VEL
LIN {X 0,Y 494.712,Z 767.588,A -85,B 0,C 180,E1 13340.396,E2 13340.396} C_VEL
LIN {X 0,Y 500.124,Z 774.698,A -85,B 0,C 180,E1 13342.021,E2 13342.021} C_VEL
LIN {X 0,Y 512.928,Z 792.267,A -85,B 0,C 180,E1 13345.47,E2 13345.47} C_VEL
LIN {X 0,Y 530.166,Z 820.106,A -85,B 0,C 180,E1 13349.75,E2 13349.75} C_VEL
LIN {X 0,Y 543.983,Z 849.212,A -85,B 0,C 180,E1 13353.314,E2 13353.314} C_VEL
LIN {X 0,Y 546.717,Z 858.661,A -85,B 0,C 180,E1 13354.236,E2 13354.236} C_VEL
LIN {X 0,Y 538.906,Z 903.26,A -85,B 0,C 180,E1 13356.22,E2 13356.22} C_VEL
LIN {X 0,Y 529.168,Z 946.579,A -85,B 0,C 180,E1 13358.928,E2 13358.928} C_VEL
LIN {X 0,Y 519.416,Z 984.076,A -85,B 0,C 180,E1 13362.053,E2 13362.053} C_VEL
LIN {X 0,Y 509.27,Z 1020.092,A -85,B 0,C 180,E1 13365.998,E2 13365.998} C_VEL
LIN {X 0,Y 500.454,Z 1050.567,A -85,B 0,C 180,E1 13370.365,E2 13370.365} C_VEL
LIN {X 0,Y 493.259,Z 1077.092,A -85,B 0,C 180,E1 13375.293,E2 13375.293} C_VEL
LIN {X 0,Y 488.021,Z 1099.248,A -85,B 0,C 180,E1 13380.812,E2 13380.812} C_VEL
LIN {X 0,Y 485.273,Z 1114.758,A -85,B 0,C 180,E1 13386.121,E2 13386.121} C_VEL
LIN {X 0,Y 483.825,Z 1125.881,A -85,B 0,C 180,E1 13391.801,E2 13391.801} C_VEL
LIN {X 0,Y 483.157,Z 1131.535,A -85,B 0,C 180,E1 13397.355,E2 13397.355} C_VEL
LIN {X 0,Y 483.277,Z 1132.296,A -85,B 0,C 180,E1 13402.816,E2 13402.816} C_VEL
LIN {X 0,Y 483.665,Z 1128.26,A -85,B 0,C 180,E1 13408.21,E2 13408.21} C_VEL
LIN {X 0,Y 484.404,Z 1120.164,A -85,B 0,C 180,E1 13413.273,E2 13413.273} C_VEL
LIN {X 0,Y 486.466,Z 1107.302,A -85,B 0,C 180,E1 13418.486,E2 13418.486} C_VEL
LIN {X 0,Y 490.597,Z 1086.747,A -85,B 0,C 180,E1 13424.266,E2 13424.266} C_VEL
LIN {X 0,Y 496.328,Z 1063.496,A -85,B 0,C 180,E1 13429.1,E2 13429.1} C_VEL
LIN {X 0,Y 504.214,Z 1034.072,A -85,B 0,C 180,E1 13433.781,E2 13433.781} C_VEL
LIN {X 0,Y 513.367,Z 999.376,A -85,B 0,C 180,E1 13437.973,E2 13437.973} C_VEL
LIN {X 0,Y 522.512,Z 962.709,A -85,B 0,C 180,E1 13441.371,E2 13441.371} C_VEL
LIN {X 0,Y 532.152,Z 919.34,A -85,B 0,C 180,E1 13444.374,E2 13444.374} C_VEL
LIN {X 0,Y 539.799,Z 877.005,A -85,B 0,C 180,E1 13446.504,E2 13446.504} C_VEL
LIN {X 0,Y 542.471,Z 854.874,A -85,B 0,C 180,E1 13447.438,E2 13447.438} C_VEL
LIN {X 0,Y 524.256,Z 816.993,A -85,B 0,C 180,E1 13451.371,E2 13451.371} C_VEL
LIN {X 0,Y 505.472,Z 785.252,A -85,B 0,C 180,E1 13455.059,E2 13455.059} C_VEL
LIN {X 0,Y 488.538,Z 761.05,A -85,B 0,C 180,E1 13458.481,E2 13458.481} C_VEL
LIN {X 0,Y 484.978,Z 755.812,A -85,B 0,C 180,E1 13459.267,E2 13459.267} C_VEL
LIN {X 0,Y 481.974,Z 750.566,A -85,B 0,C 180,E1 13459.976,E2 13459.976} C_VEL
LIN {X 0,Y 481.904,Z 749.56,A -85,B 0,C 180,E1 13460.061,E2 13460.061} C_VEL
LIN {X 0,Y 481.833,Z 749.56,A -85,B 0,C 180,E1 13465.624,E2 13465.624} C_VEL
LIN {X 0,Y 481.946,Z 749.56,A -85,B 0,C 180,E1 13471.939,E2 13471.939} C_VEL
LIN {X 0,Y 482.142,Z 749.56,A -85,B 0,C 180,E1 13477.902,E2 13477.902} C_VEL
LIN {X 0,Y 482.354,Z 749.56,A -85,B 0,C 180,E1 13483.618,E2 13483.618} C_VEL
LIN {X 0,Y 482.806,Z 749.56,A -85,B 0,C 180,E1 13489.171,E2 13489.171} C_VEL
LIN {X 0,Y 483.112,Z 749.56,A -85,B 0,C 180,E1 13494.61,E2 13494.61} C_VEL
LIN {X 0,Y 483.477,Z 749.56,A -85,B 0,C 180,E1 13499.995,E2 13499.995} C_VEL
LIN {X 0,Y 483.184,Z 749.56,A -85,B 0,C 180,E1 13505.379,E2 13505.379} C_VEL
LIN {X 0,Y 482.825,Z 749.56,A -85,B 0,C 180,E1 13510.819,E2 13510.819} C_VEL
LIN {X 0,Y 482.628,Z 749.56,A -85,B 0,C 180,E1 13516.363,E2 13516.363} C_VEL
LIN {X 0,Y 482.371,Z 749.56,A -85,B 0,C 180,E1 13522.077,E2 13522.077} C_VEL
LIN {X 0,Y 482.29,Z 750.156,A -85,B 0,C 180,E1 13525.833,E2 13525.833} C_VEL
LIN {X 0,Y 484.604,Z 755.188,A -85,B 0,C 180,E1 13526.409,E2 13526.409} C_VEL
LIN {X 0,Y 487.361,Z 758.675,A -85,B 0,C 180,E1 13527.009,E2 13527.009} C_VEL
LIN {X 0,Y 505.868,Z 785.667,A -85,B 0,C 180,E1 13530.763,E2 13530.763} C_VEL
LIN {X 0,Y 527.562,Z 820.526,A -85,B 0,C 180,E1 13534.634,E2 13534.634} C_VEL
LIN {X 0,Y 548.266,Z 859.621,A -85,B 0,C 180,E1 13538.322,E2 13538.322} C_VEL
LIN {X 0,Y 550.704,Z 864.996,A -85,B 0,C 180,E1 13538.783,E2 13538.783} C_VEL
LIN {X 0,Y 544.432,Z 911.177,A -85,B 0,C 180,E1 13540.244,E2 13540.244} C_VEL
LIN {X 0,Y 536.398,Z 957.833,A -85,B 0,C 180,E1 13542.404,E2 13542.404} C_VEL
LIN {X 0,Y 527.356,Z 1001.518,A -85,B 0,C 180,E1 13545.12,E2 13545.12} C_VEL
LIN {X 0,Y 516.983,Z 1045.458,A -85,B 0,C 180,E1 13548.737,E2 13548.737} C_VEL
LIN {X 0,Y 507.845,Z 1082.691,A -85,B 0,C 180,E1 13552.719,E2 13552.719} C_VEL
LIN {X 0,Y 499.009,Z 1118.563,A -85,B 0,C 180,E1 13557.632,E2 13557.632} C_VEL
LIN {X 0,Y 492.64,Z 1146.827,A -85,B 0,C 180,E1 13562.605,E2 13562.605} C_VEL
LIN {X 0,Y 487.836,Z 1171.427,A -85,B 0,C 180,E1 13568.178,E2 13568.178} C_VEL
LIN {X 0,Y 485.217,Z 1187.682,A -85,B 0,C 180,E1 13573.256,E2 13573.256} C_VEL
LIN {X 0,Y 484.116,Z 1196.55,A -85,B 0,C 180,E1 13577.028,E2 13577.028} C_VEL
LIN {X 0,Y 481.334,Z 1199.62,A -85,B 0,C 180,E1 13578.51,E2 13578.51} C_VEL
LIN {X 0,Y 475.779,Z 1203.375,A -85,B 0,C 180,E1 13580.75,E2 13580.75} C_VEL
LIN {X 0,Y 475.666,Z 1203.715,A -85,B 0,C 180,E1 13581.011,E2 13581.011} C_VEL
LIN {X 0,Y 475.465,Z 1208.878,A -85,B 0,C 180,E1 13586.355,E2 13586.355} C_VEL
LIN {X 0,Y 475.641,Z 1209.666,A -85,B 0,C 180,E1 13591.82,E2 13591.82} C_VEL
LIN {X 0,Y 475.589,Z 1205.911,A -85,B 0,C 180,E1 13597.301,E2 13597.301} C_VEL
LIN {X 0,Y 476.169,Z 1197.284,A -85,B 0,C 180,E1 13602.834,E2 13602.834} C_VEL
LIN {X 0,Y 477.803,Z 1184.925,A -85,B 0,C 180,E1 13607.959,E2 13607.959} C_VEL
LIN {X 0,Y 481.203,Z 1165.115,A -85,B 0,C 180,E1 13613.602,E2 13613.602} C_VEL
LIN {X 0,Y 486.54,Z 1139.809,A -85,B 0,C 180,E1 13619.031,E2 13619.031} C_VEL
LIN {X 0,Y 494.358,Z 1107.506,A -85,B 0,C 180,E1 13624.385,E2 13624.385} C_VEL
LIN {X 0,Y 503.658,Z 1071.156,A -85,B 0,C 180,E1 13629.054,E2 13629.054} C_VEL
LIN {X 0,Y 513.99,Z 1031.174,A -85,B 0,C 180,E1 13633.104,E2 13633.104} C_VEL
LIN {X 0,Y 525.102,Z 985.743,A -85,B 0,C 180,E1 13636.604,E2 13636.604} C_VEL
LIN {X 0,Y 534.905,Z 940.813,A -85,B 0,C 180,E1 13639.191,E2 13639.191} C_VEL
LIN {X 0,Y 542.77,Z 896.524,A -85,B 0,C 180,E1 13641.059,E2 13641.059} C_VEL
LIN {X 0,Y 546.527,Z 867.428,A -85,B 0,C 180,E1 13642.038,E2 13642.038} C_VEL
LIN {X 0,Y 532.324,Z 835.034,A -85,B 0,C 180,E1 13645.366,E2 13645.366} C_VEL
LIN {X 0,Y 516.492,Z 808.338,A -85,B 0,C 180,E1 13648.983,E2 13648.983} C_VEL
LIN {X 0,Y 499.806,Z 784.265,A -85,B 0,C 180,E1 13653.278,E2 13653.278} C_VEL
LIN {X 0,Y 489.34,Z 770.523,A -85,B 0,C 180,E1 13656.517,E2 13656.517} C_VEL
LIN {X 0,Y 484.47,Z 763.9,A -85,B 0,C 180,E1 13658.265,E2 13658.265} C_VEL
LIN {X 0,Y 480.466,Z 758.552,A -85,B 0,C 180,E1 13659.85,E2 13659.85} C_VEL
LIN {X 0,Y 478.88,Z 756.654,A -85,B 0,C 180,E1 13660.516,E2 13660.516} C_VEL
LIN {X 0,Y 474.892,Z 751.953,A -85,B 0,C 180,E1 13662.33,E2 13662.33} C_VEL
LIN {X 0,Y 474.54,Z 749.56,A -85,B 0,C 180,E1 13662.805,E2 13662.805} C_VEL
LIN {X 0,Y 474.913,Z 749.56,A -85,B 0,C 180,E1 13668.999,E2 13668.999} C_VEL
LIN {X 0,Y 475.253,Z 749.56,A -85,B 0,C 180,E1 13674.531,E2 13674.531} C_VEL
LIN {X 0,Y 475.561,Z 749.56,A -85,B 0,C 180,E1 13680.005,E2 13680.005} C_VEL
LIN {X 0,Y 475.183,Z 749.56,A -85,B 0,C 180,E1 13685.48,E2 13685.48} C_VEL
LIN {X 0,Y 474.884,Z 749.56,A -85,B 0,C 180,E1 13691.012,E2 13691.012} C_VEL
LIN {X 0,Y 474.703,Z 750.07,A -85,B 0,C 180,E1 13692.996,E2 13692.996} C_VEL
LIN {X 0,Y 476.646,Z 754.83,A -85,B 0,C 180,E1 13694.05,E2 13694.05} C_VEL
LIN {X 0,Y 480.545,Z 758.331,A -85,B 0,C 180,E1 13695.684,E2 13695.684} C_VEL
LIN {X 0,Y 484.134,Z 763.643,A -85,B 0,C 180,E1 13697.138,E2 13697.138} C_VEL
LIN {X 0,Y 486.319,Z 766.165,A -85,B 0,C 180,E1 13697.933,E2 13697.933} C_VEL
LIN {X 0,Y 492.59,Z 774.683,A -85,B 0,C 180,E1 13700.078,E2 13700.078} C_VEL
LIN {X 0,Y 502.224,Z 787.717,A -85,B 0,C 180,E1 13702.974,E2 13702.974} C_VEL
LIN {X 0,Y 517.306,Z 810.449,A -85,B 0,C 180,E1 13707.045,E2 13707.045} C_VEL
LIN {X 0,Y 532.12,Z 837.78,A -85,B 0,C 180,E1 13710.925,E2 13710.925} C_VEL
LIN {X 0,Y 541.258,Z 859.991,A -85,B 0,C 180,E1 13713.553,E2 13713.553} C_VEL
LIN {X 0,Y 533.46,Z 904.98,A -85,B 0,C 180,E1 13715.637,E2 13715.637} C_VEL
LIN {X 0,Y 523.176,Z 949.058,A -85,B 0,C 180,E1 13718.431,E2 13718.431} C_VEL
LIN {X 0,Y 513.06,Z 986.247,A -85,B 0,C 180,E1 13721.596,E2 13721.596} C_VEL
LIN {X 0,Y 502.532,Z 1022.097,A -85,B 0,C 180,E1 13725.591,E2 13725.591} C_VEL
LIN {X 0,Y 492.885,Z 1053.968,A -85,B 0,C 180,E1 13730.299,E2 13730.299} C_VEL
LIN {X 0,Y 485.704,Z 1079.073,A -85,B 0,C 180,E1 13735.139,E2 13735.139} C_VEL
LIN {X 0,Y 480.253,Z 1101.176,A -85,B 0,C 180,E1 13740.811,E2 13740.811} C_VEL
LIN {X 0,Y 477.401,Z 1116.348,A -85,B 0,C 180,E1 13746.258,E2 13746.258} C_VEL
LIN {X 0,Y 476.011,Z 1126.31,A -85,B 0,C 180,E1 13751.492,E2 13751.492} C_VEL
LIN {X 0,Y 475.305,Z 1132.111,A -85,B 0,C 180,E1 13757.142,E2 13757.142} C_VEL
LIN {X 0,Y 475.382,Z 1132.971,A -85,B 0,C 180,E1 13762.696,E2 13762.696} C_VEL
LIN {X 0,Y 475.814,Z 1129.095,A -85,B 0,C 180,E1 13768.181,E2 13768.181} C_VEL
LIN {X 0,Y 476.529,Z 1122.071,A -85,B 0,C 180,E1 13772.836,E2 13772.836} C_VEL
LIN {X 0,Y 478.726,Z 1108.383,A -85,B 0,C 180,E1 13778.624,E2 13778.624} C_VEL
LIN {X 0,Y 482.737,Z 1089.128,A -85,B 0,C 180,E1 13784.21,E2 13784.21} C_VEL
LIN {X 0,Y 488.545,Z 1066.752,A -85,B 0,C 180,E1 13789.066,E2 13789.066} C_VEL
LIN {X 0,Y 497.149,Z 1035.631,A -85,B 0,C 180,E1 13794.14,E2 13794.14} C_VEL
LIN {X 0,Y 506.321,Z 1002.235,A -85,B 0,C 180,E1 13798.268,E2 13798.268} C_VEL
